DATA_BLOCK "FLT"   // DB142
{ S7_Optimized_Access := 'FALSE' }
VERSION : 0.0
// --------------------------------------------------------------------------------
//     program     :    FLT
//     description :    FLT signals       
//     name        :    G. Eibelshaeuser
//     date        :    26.10.2007
// 
//     revision    :
//     name        :
//     date        :    
//                     (c)PVA TePla AG       
//     --------------------------------------------------------------------------------
   VAR
      PD_TIME_10MBAR : Bool;   // F001 pump down time to 10 mbar exceeded
      PD_TIME_1MBAR : Bool;   // F002 pump down time to 1 mbar exceeded
      PD_TIME_01MBAR : Bool;   // F003 pump down time to 0,1 mabar exceeded
      PD_TIME_005MBAR : Bool;   // F004 pump down time to 0,05 mbar exceeded
      PD_TIME_FINAL : Bool;   // F005 pump down time to final pressure exceeded
      PD_LEAKTEST : Bool;   // F006 leaktest failed
      PD_GATE_VALVE_CLOSED : Bool;   // F007 gate valve is closed
      ME_CR_REF_POS_NOT_FND : Bool;   // F008 crucible reference position not found
      ME_LEAK_TST_FDR : Bool;   // F009 leaktest feeder failed
      ME_PRS_DROP_FDR : Bool;   // F010 pressure drop feeder too high
      ME_SPARE_F011 : Bool;   // F011
      DI_IMAGE_TO_DARK : Bool;   // F012 image too dark for dipping
      DI_TIME_CAM_EXCEEDED : Bool;   // F013 time till seed detection exceeded
      DI_TIME_MELT_EXCEEDED : Bool;   // F014 time till melt contact exceeded
      DI_SEED_NOT_CAM_STOPPED : Bool;   // F015 seed not cam. stopped before dipping
      DI_MCC_ERROR_1 : Bool;   // F016 melt contact control function error
      DI_MCC_ERROR_2 : Bool;   // F017 melt contact control input error
      DI_ISOLATION_FAULT : Bool;   // F018 crystal drive unit not isolated from ground
      DI_SPARE_F019 : Bool;   // F019
      DI_SPARE_F020 : Bool;   // F020
      NE_MAX_LEN : Bool;   // F021 max. neck length reached without constant diameter
      NE_SPARE_F022 : Bool;   // F022
      SH_MLT_LVL_SFT : Bool;   // F023 invalid melt level shift parameter in phase shoulder
      SH_SPARE_F024 : Bool;   // F024
      BY_SPARE_F025 : Bool;   // F025
      BY_SPARE_F026 : Bool;   // F026
      EC_XT_OUT_OF_MELT : Bool;   // F027 crystal out of melt
      EC_SPARE_F028 : Bool;   // F028
      EC_SPARE_F029 : Bool;   // F029
      RE_SPARE_F030 : Bool;   // F030
      RE_SPARE_F031 : Bool;   // F031
      SD_SMALL_DIS_XT_CR : Bool;   // F032 distance between crystal and crucible too small
      FDR_NOT_IN_HOME_POS : Bool;   // F033 feeder is not in home position
      CR_ROT_OSCI : Bool;   // F034 frequency of cruc. rot. oscillation too high out of range faults
      XT_ROT_OUT_OF_RNG : Bool;   // F035 crystal rotation out of range
      XT_LFT_OUT_OF_RNG : Bool;   // F036 crystal lift out of range
      CR_ROT_OUT_OF_RNG : Bool;   // F037 crucible rotation out of range
      CR_LFT_OUT_OF_RNG : Bool;   // F038 crucible lift out of range
      GAS_FLW_1_OUT_OF_RNG : Bool;   // F039 gas flow 1 out of range
      GAS_FLW_2_OUT_OF_RNG : Bool;   // F040 gas flow 2 out of range
      PRS_OUT_OF_RNG : Bool;   // F041 pressure out of range
      HTR_1_PWR_OUT_OF_RNG : Bool;   // F042 main heater power out of range
      HTR_2_PWR_OUT_OF_RNG : Bool;   // F043 bottom heater power out of range
      NECK_DIA_BELOW_LIMIT : Bool;   // F044 neck diameter below limit
      XT_GROWTH_OUT_OF_RNG : Bool;   // F045 crystal growth out of range
      XT_DIA_OUT_OF_RNG : Bool;   // F046 crystal diameter out of range
      AVG_PULL_SPD_OUT_OF_RNG : Bool;   // F047 average pull speed out of range
      MELT_LEVEL_OUT_OF_RNG : Bool;   // F048 melt level out of range
      HTR_1_RES_OUT_OF_RNG : Bool;   // F049 resistance change main heater out of range
      HTR_2_RES_OUT_OF_RNG : Bool;   // F050 resistance change bottom heater out of range
      MAG_1_CUR_OUT_OF_RNG : Bool;   // F051 magnet current coil 1 out of range
      MAG_2_CUR_OUT_OF_RNG : Bool;   // F052 magnet current coil 2 out of range
      CAM_THR_RATIO : Bool;   // F053 threshold ratio out of range from recipe temperature switches
      WTR_TMP_CUR_FEED : Bool;   // F054 water temp. current feed through heater 1
      HTR_2_TAS_CUR_FEED : Bool;   // F055 water temp. current feed through heater 2
      WTR_TMP_CR_SFT : Bool;   // F056 water temp. crucible shaft
      WTR_TMP_PWR_CAB : Bool;   // F057 water temp. high current cables
      WTR_TMP_GCH : Bool;   // F058 water temp. gate chamber
      CHAMBERS_TAS : Bool;   // F059 water temp. chambers
      VIP_TAS : Bool;   // F060 water temp. view ports
      XT_TAS : Bool;   // F061 water temp. xtal shaft
      EXH_TAS : Bool;   // F062 water temp. exhaust
      SPARE_F063 : Bool;   // F063 water flow switches -------------------
      SPARE_F064 : Bool;   // F064 spare
      WTR_FLW_HTR_1 : Bool;   // F065 water flow heater power supply
      WTR_FLW_GCH : Bool;   // F066 water flow gate chamber
      WTR_FLW_CR_SFT : Bool;   // F067 water flow crucible shaft
      XT_WFS : Bool;   // F068 water flow xtal shaft heater alarm -------------------
      HTR_SCR_WRN : Bool;   // F069 heater rectifier temp warning
      HTR_SCR_ALM : Bool;   // F070 heater rectifier temp alarm
      HTR_TRF_WRN : Bool;   // F071 heater transformer temp warning
      HTR_TRF_ALM : Bool;   // F072 heater transformer temp alarm
      THY_CTRL_1_OV_LD : Bool;   // F073 thyristor controller heater 1 overload
      THY_CTRL_1_HI_TMP : Bool;   // F074 thyristor controller heater 1 high temperature
      THY_CTRL_1_ER : Bool;   // F075 thyristor controller heater 1 fault
      HTR_2_OVERCURRENT : Bool;   // F076 heater 2 overcurrent
      HTR_2_CUR_LIMIT : Bool;   // F077 heater 2 current limit active
      HTR_2_ITL : Bool;   // F078 heater 2 interlock active UPS alarm ---------
      UPS_24V_ALM : Bool;   // F079 24 V UPS error
      UPS_24V_SPL_MIS : Bool;   // F080 24 V supply for UPS failed
      THY_CTRL_1_OV_VLT : Bool;   // F081 thryristor controller heater 1 over voltage
      CB_FLT_COMP_400V : Bool;   // F082 circuit breaker fault AC 400V compensation
      TMP_MAIN_CBT : Bool;   // F083 temperature fault main cabinet +K1 breakers and fuses ------------------
      CB_FLT_DC24V : Bool;   // F084 circuit breaker fault DC 24 V
      CB_FLT_AC230V : Bool;   // F085 circuit breaker fault AC 230 V
      CB_FLT_DRV : Bool;   // F086 circuit breaker fault drive units
      CB_FLT_AC400V : Bool;   // F087 circuit breaker fault AC 400V
      MAIN_SWITCH_OFF : Bool;   // F088 main switch of plant is off
      HTR_1_OVERCURRENT : Bool;   // F089 heater 1 overcurrent
      HTR_1_CUR_LIMIT : Bool;   // F090 heater 1 current limit active
      HTR_1_ITL : Bool;   // F091 heater 1 interlock active
      HTR_WFS : Bool;   // F092 water flow heater
      CGT_WFS : Bool;   // F093 water flow gate chamber
      CR_WFS : Bool;   // F094 water flow crucible shaft safety limit switches ---------------------
      XT_TOP_POS : Bool;   // F095 safty limit switch seed chuck in highest pos.
      XT_SLS : Bool;   // F096 safty limit switch crystal lift
      CR_SLS : Bool;   // F097 safty limit switch crucible lift
      CHAMBER_SLS : Bool;   // F098 safty limit switch chamber lift
      MAG_SLS : Bool;   // F099 safty limit switch magnet lift
      MAIN_LINE_460V_OFF : Bool;   // F100 460V main power supply is off image processing unit ---------------------
      INIT_FLT_IM_PROC_UNIT : Bool;   // F101 initialisation fault image processing unit
      INV_DATA_IM_PROC_UNIT : Bool;   // F102 invalid data from image processing unit
      CAM_INTERFACE_INIT : Bool;   // F103 camera serial interface init failed
      CAM_THR_ADJ_STOPPED : Bool;   // F104 automatic threshold adjustment interrupted
      CAM_THR_ADJ_ABORTED : Bool;   // F105 automatic threshold adjustment aborted common ------
      MAIN_LINE_OFF : Bool;   // F106 main power supply is off
      COM_AIR_PRS_LOW : Bool;   // F107 compressed air pressure is below limit
      PLC_INIT_FLT_NO_RECIPE : Bool;   // F108 no recipe in PLC
      EMO : Bool;   // F109 emergency off
      DRV_CAL_MIS : Bool;   // F110 drive calibration is missing
      LSR_RCV : Bool;   // F111 laser receiver detects no beam drive controller faults
      DRV_XT_LFT_PAR_FLT : Bool;   // F112 parameter fault drive controller crystal lift
      DRV_XT_LFT_RUN_FLT : Bool;   // F113 operating fault drive controller crystal lift
      DRV_XT_ROT_PAR_FLT : Bool;   // F114 parameter fault drive controller crystal rotation
      DRV_XT_ROT_RUN_FLT : Bool;   // F115 operating fault drive controller crystal rotation
      DRV_CR_LFT_PAR_FLT : Bool;   // F116 parameter fault drive controller crucible lift
      DRV_CR_LFT_RUN_FLT : Bool;   // F117 operating fault drive controller crucible lift
      DRV_CR_ROT_PAR_FLT : Bool;   // F118 parameter fault drive controller crucible rotation
      DRV_CR_ROT_RUN_FLT : Bool;   // F119 operating fault drive controller crucible rotation
      DRV_CHB_LFT_PAR_FLT : Bool;   // F120 parameter fault drive controller chamber lift
      DRV_CHB_LFT_RUN_FLT : Bool;   // F121 operating fault drive controller chamber lift
      DRV_CHB_SW_PAR_FLT : Bool;   // F122 parameter fault drive controller chamber swivel
      DRV_CHB_SW_RUN_FLT : Bool;   // F123 operating fault drive controller chamber swivel
      SPARE_F124 : Bool;   // F124
      WTR_TMP_CFT_2 : Bool;   // F125 water temperature current feed throughs 2
      WTR_TMP_GATE : Bool;   // F126 water temperature gate and gate valve
      WTR_TMP_SPC : Bool;   // F127 water temperature spacer and view ports
      WTR_TMP_VSL : Bool;   // F128 water temperature vessel parts Vacuum faults --------------------
      P1 : Bool;   // F129 vacuum pump 1 not ready
      P2 : Bool;   // F130 vacuum pump 2 not ready
      P3 : Bool;   // F131 vacuum pump 3 not ready
      P1_TMP_HIGH : Bool;   // F132 temperature fault of pump 1
      P2_TMP_HIGH : Bool;   // F133 temperature fault of pump 2
      P3_TMP_HIGH : Bool;   // F134 temperature fault of pump 3
      V7 : Bool;   // F135 undefined position gate valve
      V2_1 : Bool;   // F136 vacuum valve V2.1 not open
      V2_2 : Bool;   // F137 vacuum valve V2.2 not open
      V3 : Bool;   // F138 vacuum valve V3 not open
      WTR_TMP_FCH : Bool;   // F139 water temperature furnace chamber
      WTR_TMP_TCH : Bool;   // F140 water temperature top chamber
      P1_SP_WRN : Bool;   // F141 vacuum pump 1 warning active
      FDR_HOP_NOT_CON : Bool;   // F142 hopper not connected to feeder
      P3_SP_WRN : Bool;   // F143 vacuum pump 3 warning active
      WTR_FLW_FCH : Bool;   // F144 water flow furnace chamber
      WTR_FLW_TCH : Bool;   // F145 water flow top chamber
      WTR_FLW_CFT_2 : Bool;   // F146 water flow current feed throughs 2
      WTR_FLW_GATE : Bool;   // F147 water flow gate and gate valve
      WTR_FLW_SPC : Bool;   // F148 water flow spacer and view ports
      WTR_FLW_VSL : Bool;   // F149 water flow bottom chamber Position encoder faults -----------------------
      ENC_XT_LFT : Bool;   // F150 position error crystal lift
      ENC_CR_LFT : Bool;   // F151 position error crucible lift
      ENC_CGT_LFT : Bool;   // F152 position error handling lift
      SPARE_F153 : Bool;   // F153 image processing with DVT Cam -----------------------------
      CAM_ROI_OUTSIDE : Bool;   // F154 camera measurement area is outside the image frame
      DVT_PRD_NO_PLC : Bool;   // F155 Produktnummer in der SPS ung黮tig
      DVT_PRD_NO_IMG_SEN : Bool;   // F156 Produktnummer in Kamera ist ung黮tig
      CAM_COM_SEND : Bool;   // F157 Sendefehler SPS - Kamera
      CAM_DATA_RECV : Bool;   // F158 Empfangsfehler SPS - Kamera
      DVT_NO_PRD : Bool;   // F159 kein "P" im Telegramm von Kamera
      DVT_DATA_MSG : Bool;   // F160 Daten von Kamera sind ung黮tig
      DVT_PRD_NO_DIF : Bool;   // F161 Produktnummer von Kamera ist falsch
      CAM_NDR_TOUT : Bool;   // F162 keine Daten von Kamera empfangen
      DVT_IMG_SEN : Bool;   // F163 Bildverarbeitung von Kamera gescheitert
      CAM_NO_CTR_FND : Bool;   // F164 Kamera findet keinen messbaren Kontrast
      CAM_MSR_INSTAB : Bool;   // F165 Meniskusmessung instabil, Fehlmessungen -----------------------
      V7_CLOSED : Bool;   // F166 gate valve closed (crystal down disabled)
      CLF_CLP_POS : Bool;   // F167 undefined position furnace clamp
      CGT_COUPLE : Bool;   // F168 undefined position coupling gate/furnace
      CLF_SWL_POS : Bool;   // F169 undefined position lower furnace
      HND_VACUUM : Bool;   // F170 furnace is not vented !
      CLF_CLAMP : Bool;   // F171 upper furnace is not connected with gate !
      XT_FORK : Bool;   // F172 safety fork installed (crystal down disabled)
      SEED_TMP : Bool;   // F173 seed chuck is too hot; crystal lift stopped
      FDR_TUBE_TME_OUT : Bool;   // F174 feeding tube did not reach end position
      GCH_NOT_CL : Bool;   // F175 gate chamber not closed
      CR_ROT_CAL : Bool;   // F176 calibration fault crucible rotation drive
      CR_LFT_CAL : Bool;   // F177 calibration fault crucible lift drive
      XT_ROT_CAL : Bool;   // F178 calibration fault crystal rotation drive
      XT_LFT_CAL : Bool;   // F179 calibration fault crystal lift drive
      WTR_FLW_PLT : Bool;   // F180 water flow chamber parts and view ports
      PWR_SPL_WFS : Bool;   // F181 water flow heater power supply
      WTR_FLW_CUR_FEED : Bool;   // F182 water flow current feed through heater 1
      WTR_FLW_PWR_CAB : Bool;   // F183 water flow high current cables
      WTR_FLW_GCH_V : Bool;   // F184 water flow gate chamber valve
      WTR_FLW_CONE : Bool;   // F185 water flow cone alarm /nur SC22 AUO)
      WTR_TMP_PLT : Bool;   // F186 water temp. chamber parts and view ports
      WTR_TMP_GCH_V : Bool;   // F187 water temp. gate chamber valve
      WTR_TMP_HTR_1 : Bool;   // F188 water temp. heater power supply
      PWR_SPL_INT_TAS : Bool;   // F189 water temp. transformer intern
      WTR_TMP_HIGH_LIM : Bool;   // F190 water temp. high limit reached
      HTR_PWR_CAB_TAS : Bool;   // F191 water temp. high power cables
      HTR_1_TAS_CUR_FEED : Bool;   // F192 water temp. current feed through heater 1
      CGT_TAS : Bool;   // F193 water temp. gate chamber
      CR_TAS : Bool;   // F194 water temp. crucible shaft MAGNET FAULTS -------------
      MAG_1_RES_OUT_OF_RNG : Bool;   // F195 resistance change upper magnet out of range
      MAG_2_RES_OUT_OF_RNG : Bool;   // F196 resistance change lower magnet out of range
      MAG_WFS : Bool;   // F197 water flow magnet power supply intern
      MAG_1_ITL : Bool;   // F198 magnet 1 rectifier interlock active
      MAG_2_ITL : Bool;   // F199 magnet 2 rectifier interlock active
      MAG_TMP_ALM : Bool;   // F200 magnet transformer temperature alarm
      MAG_1_EXT_ITL : Bool;   // F201 external interlock magnet 1
      MAG_2_EXT_ITL : Bool;   // F202 external interlock magnet 2
      MAG_DOOR_ITL : Bool;   // F203 door interlock magnet power supply
      MAG_1_OVERCURRENT : Bool;   // F204 magnet 1 overcurrent
      MAG_2_OVERCURRENT : Bool;   // F205 magnet 2 overcurrent
      PAR_FLT_MAG_1_CUR : Bool;   // F206 magnet 1 current setpoint out of range
      PAR_FLT_MAG_2_CUR : Bool;   // F207 magnet 2 current setpoint out of range
      MAG_LFT_SDL_ERR : Bool;   // F208 Magnet lift error - upward lift disabled
      MAG_TAS : Bool;   // -----------------
      DP_ADR_08_NOT_PRESENT : Bool;   // F210 dp-slave not present (+N2)
      DP_ADR_09_NOT_PRESENT : Bool;   // F211 dp-slave not present (+R1.B1)
      DP_ADR_10_NOT_PRESENT : Bool;   // F212 dp-slave not present (+N1)
      DP_ADR_11_NOT_PRESENT : Bool;   // F213 dp-slave not present (+N4)
      DP_ADR_16_NOT_PRESENT : Bool;   // F214 dp-slave encoder crystal lift not present
      DP_ADR_17_NOT_PRESENT : Bool;   // F215 dp-slave encoder crucible lift not present
      DP_ADR_18_NOT_PRESENT : Bool;   // F216 dp-slave encoder handling lift not present
      DP_ADR_32_NOT_PRESENT : Bool;   // F217 dp-slave controller crystal rot. not present
      DP_ADR_33_NOT_PRESENT : Bool;   // F218 dp-slave controller crystal lift not present
      DP_ADR_34_NOT_PRESENT : Bool;   // F219 dp-slave controller crucible rot. not present
      DP_ADR_35_NOT_PRESENT : Bool;   // F220 dp-slave controller crucible lift not present
      DP_ADR_36_NOT_PRESENT : Bool;   // F221 dp-slave controller gate swinging not present
      DP_ADR_37_NOT_PRESENT : Bool;   // F222 dp-slave controller gate lifting not present
      DP_ADR_40_NOT_PRESENT : Bool;   // F223 dp-slave main heater not present
      DP_ADR_41_NOT_PRESENT : Bool;   // F224 dp-slave botton heater not present
      DP_ADR_45_NOT_PRESENT : Bool;   // F225 dp-slave magnet coil 1 not present
      DP_ADR_46_NOT_PRESENT : Bool;   // F225 dp-slave magnet coil 2 not present
      DP_ADR_64_NOT_PRESENT : Bool;   // F227 dp-slave not present (+N5)
      DP_ADR_13_NOT_PRESENT : Bool;   // F228 dp-slave not present (+N3)
      DP_ADR_48_NOT_PRESENT : Bool;   // F229 dp-slave MFC 1 not present
      DP_ADR_42_NOT_PRESENT : Bool;   // F230 dp-slave SCR controller heater 1 not present
      DP_ADR_43_NOT_PRESENT : Bool;   // F231 dp-slave SCR controller heater 2 not present
      DP_ADR_38_NOT_PRESENT : Bool;   // F232 dp_slave pump unit not present
      DP_ADR_08_ERROR : Bool;   // F233 dp-slave fault (+N1)
      DP_ADR_09_ERROR : Bool;   // F234 dp-slave fault (+R1.B1)
      DP_ADR_10_ERROR : Bool;   // F235 dp-slave fault (+N2)
      DP_ADR_11_ERROR : Bool;   // F236 dp-slave fault (+N4)
      DP_ADR_16_ERROR : Bool;   // F237 dp-slave encoder crystal lift fault
      DP_ADR_17_ERROR : Bool;   // F238 dp-slave encoder crucible lift fault
      DP_ADR_18_ERROR : Bool;   // F239 dp-slave encoder handling lift fault
      DP_ADR_32_ERROR : Bool;   // F240 dp-slave controller crystal rot. fault
      DP_ADR_33_ERROR : Bool;   // F241 dp-slave controller crystal lift fault
      DP_ADR_34_ERROR : Bool;   // F242 dp-slave controller crucible rot. fault
      DP_ADR_35_ERROR : Bool;   // F243 dp-slave controller crucible lift fault
      DP_ADR_36_ERROR : Bool;   // F244 dp-slave controller gate swinging fault
      DP_ADR_37_ERROR : Bool;   // F245 dp-slave controller gate lifting fault
      DP_ADR_40_ERROR : Bool;   // F246 dp-slave main heater fault
      DP_ADR_41_ERROR : Bool;   // F247 dp-slave bottom heater fault
      DP_ADR_45_ERROR : Bool;   // F248 dp-slave magnet coil 1 fault
      DP_ADR_46_ERROR : Bool;   // F249 dp-slave magnet coil 2 fault
      DP_ADR_64_ERROR : Bool;   // F250 dp-slave fault (+N5)
      DP_ADR_13_ERROR : Bool;   // F251 dp-slave fault (+N3)
      DP_ADR_48_ERROR : Bool;   // F252 dp-slave MFC 1 fault
      DP_ADR_42_ERROR : Bool;   // F253 dp-slave SCR controller heater 1 fault
      DP_ADR_43_ERROR : Bool;   // F254 dp-slave SCR controller heater 2 fault
      DP_ADR_38_ERROR : Bool;   // F255 dp-slave pump unit fault
      SPARE_F256 : Bool;   // F256 device faults -------------
      MSR_WTR_TMP_PWR_CAB : Bool;   // F257 measurement water temp. high current cables
      MSR_WTR_FLW_PWR_CAB : Bool;   // F258 measurement water flow high current cables
      MSR_WTR_TMP_CUR_FEED : Bool;   // F259 measurement water temp. cur. feed through 1
      MSR_WTR_FLW_CUR_FEED : Bool;   // F260 measurement water flow cur. feed through 1
      MSR_WTR_TMP_CR_SFT : Bool;   // F261 measurement water temp. crucible shaft
      MSR_WTR_FLW_CR_SFT : Bool;   // F262 measurement water flow crucible shaft
      MSR_WTR_TMP_HTR_1 : Bool;   // F263 measurement water temp. heater 1 power supply
      MSR_WTR_FLW_HTR_1 : Bool;   // F264 measurement water flow heater 1 power supply
      MSR_WTR_TMP_CFT_2 : Bool;   // F265 measurement water temp. cur.feed through 2
      MSR_WTR_FLW_CFT_2 : Bool;   // F266 measurement water flow cur. feed through 2
      MSR_WTR_TMP_GATE : Bool;   // F267 measurement water temp. gate and gate valve
      MSR_WTR_FLW_GATE : Bool;   // F268 measurement water flow gate and gate valve
      MSR_WTR_TMP_SPC : Bool;   // F269 measurement water temp. spacer and view ports
      MSR_WTR_FLW_SPC : Bool;   // F270 measurement water flow spacer and view ports
      MSR_WTR_TMP_VSL : Bool;   // F271 measurement water temp. bottom chamber
      MSR_WTR_FLW_VSL : Bool;   // F272 measurement water flow bottom chamber
      MSR_WTR_TMP_FCH : Bool;   // F273 measurement water temp. furnace chamber
      MSR_WTR_FLW_FCH : Bool;   // F274 measurement water flow furnace chamber
      MSR_WTR_TMP_TCH : Bool;   // F275 measurement water temp. top chamber
      MSR_WTR_FLW_TCH : Bool;   // F276 measurement water flow top chamber
      MSR_ACT_MLT_TMP : Bool;   // F277 measurement melt temperature
      MSR_ACT_HTR_1_TMP : Bool;   // F278 measurement heater 1 temperature
      MLT_TMP_SIG : Bool;   // F279 melt temperature signal not valid
      HTR_1_TMP_SIG : Bool;   // F280 heater 1 temperature signal not valid
      MSR_P1_VIB : Bool;   // F281 measurement screw pump P1 vibration
      V25 : Bool;   // F282 fault valve 25
      XT_DRP_OUT_PRT_OP : Bool;   // F283 crystal drop out protection not opened
      XT_DRP_OUT_PRT_CL : Bool;   // F284 crystal drop out protection not closed
      HTR_1_SCR_ALM : Bool;   // F285 heater 1 rectifier temp alarm
      HTR_1_TRF_WRN : Bool;   // F286 heater 1 transformer temp warning
      HTR_1_TRF_ALM : Bool;   // F287 heater 1 transformer temp alarm
      HTR_2_SCR_ALM : Bool;   // F288 heater 2 rectifier temp alarm
      HTR_2_TRF_WRN : Bool;   // F289 heater 2 transformer temp warning
      HTR_2_TRF_ALM : Bool;   // F290 heater 2 transformer temp alarm
      THY_CTRL_2_OV_LD : Bool;   // F291 thyristor controller heater 2 overload
      THY_CTRL_2_HI_TMP : Bool;   // F292 thyristor controller heater 2 high temperature
      THY_CTRL_2_ER : Bool;   // F293 thyristor controller heater 2 fault
      THY_CTRL_2_OV_VLT : Bool;   // F294 thryristor controller heater 2 over voltage
      MSR_WTR_TMP_PLT : Bool;   // F295 measurement water temp. vessel and view ports
      MSR_WTR_FLW_PLT : Bool;   // F296 measurement water flow vessel and view ports
      MSR_WTR_TMP_GCH : Bool;   // F297 measurement water temp. gate chamber
      MSR_WTR_FLW_GCH : Bool;   // F298 measurement water flow gate chamber
      MSR_WTR_TMP_GCH_V : Bool;   // F299 measurement water temp. gate chamber valve
      MSR_WTR_FLW_GCH_V : Bool;   // F300 measurement water flow gate chamber valve
      V15 : Bool;   // F301 fault valve 15
      V14 : Bool;   // F302 fault valve 14
      V12 : Bool;   // F303 fault valve 12
      V18 : Bool;   // F304 fault valve 18
      V17 : Bool;   // F305 fault valve 17
      V13 : Bool;   // F306 fault valve 13
      P1_GEAR_OIL_TMP_WRN : Bool;   // F307 warning gear oil temperature of screw pump P1
      P1_GEAR_OIL_TMP_ALM : Bool;   // F308 alarm gear oil temperature of screw pump P1
      P1_COOLANT_TMP_WRN : Bool;   // F309 warning coolant temperature of screw pump P1
      P1_COOLANT_TMP_ALM : Bool;   // F310 alarm coolant temperature of screw pump P1
      DP_ADR_50_NOT_PRESENT : Bool;   // F311 dp_slave Simocode P1 not present
      DP_ADR_51_NOT_PRESENT : Bool;   // F312 dp_slave Simocode P2 not present
      DP_ADR_50_ERROR : Bool;   // F313 dp-slave Simocode P1 fault
      DP_ADR_51_ERROR : Bool;   // F314 dp-slave Simocode P2 fault
      FSH_MAIN_SI_FIL : Bool;   // F315 flushing of main Si filter not done
      FSH_AUX_SI_FIL : Bool;   // F316 flushing of aux Si filter not done
      WTR_TMP_VPTS : Bool;   // F317 water temperature view ports
      WTR_FLW_VPTS : Bool;   // F318 water flow view ports
      P1_VIB_ALM : Bool;   // F319 vibration of Pump 1 above alarm level
      MSR_P1_PT100_GEAR_OIL : Bool;   // F320 measurement error of PT100 sensor P1 gear oil temp.
      MSR_P1_PT100_COOLANT : Bool;   // F321 measurement error of PT 100 sensor P1 coolant temp.
      INIT_KL_3202 : Bool;   // F322 Initialisation of PT 100 terminal failed (KL3202)
      MSR_WTR_TMP_VPTS : Bool;   // F323 measurement water temperature view ports
      MSR_WTR_FLW_VPTS : Bool;   // F324 measurement water flow view ports
      PHA_CUR_P1 : Bool;   // F325 phase current of Pump 1 above limit
      PHA_CUR_P2 : Bool;   // F326 phase current of Pump 2 above limit
      CR_LFT_NO_ROT : Bool;   // F327 crucible lift without shaft rotation
      INGOT_ID_TIME_OUT : Bool;   // F328 timeout ingot ID
      CARRIER_ID_REFUSED : Bool;   // F329 carrier ID refused from MES
      XT_ORB_ABV_LIM : Bool;   // F330 crystal orbiting is above limit
      PU_WRN : Bool;   // F331 pump unit warning
      PU_ERR : Bool;   // F332 pump unit error
      DST_MLT_FNL_SML : Bool;   // F333 distance melt level to funnel too small
      DST_MLT_FNL_LRG : Bool;   // F334 distance metl level to funnel too large
      MLT_LVL_MSR_NOT_VALID : Bool;   // F335 melt level measurements not valid - control loop switched off
      XT_LFT_SW_LIMIT : Bool;   // F336 software limitation of crystal lift is reached
      CR_LFT_SW_LIMIT : Bool;   // F337 software limitation of crucible lift is reached
      HTR_1_PWR_SPL : Bool;   // F338 heater 1 power supply fault
      HTR_1_PWR_SPL_WRN : Bool;   // F339 heater 1 power supply warning
      HTR_1_PWR_SPL_IN_LOC : Bool;   // F340 heater 1 power supply in local operation mode
      MSR_CGT_BAR_ACT_PRS_1000 : Bool;   // F341 measurement vacuum gauge gate chamber
      OV_VLT_PRT : Bool;   // F342 over-voltage protection fault in main line
      HTR_1_BUS_BAR_TMP : Bool;   // F343 high bus bar temperature of heater 1 power supply
      HTR_2_BUS_BAR_TMP : Bool;   // F344 high bus bar temperature of heater 2 power supply
      MSR_WTR_FLW_PU : Bool;   // F345 measurement water flow pump unit
      MSR_WTR_TMP_PU : Bool;   // F346 measurement water temperature pump unit
      CAM_DI_XT_DN_ARB : Bool;   // F347 camera controlled seed down off - crystal speed reduced
      CAM_HTR_1_IN_SMI : Bool;   // F348 growth control off - heater 1 switched to semi automatic
      CAM_CRUC_ROT_IN_SMI : Bool;   // F349 growth control off - crucible rotation switched to semi automatic
      CAM_DIA_CTRL_OFF : Bool;   // F350 diameter control off - crystal lift switched to semi automatic
      WTR_TMP_PU : Bool;   // F351 water temperature pump unit
      SI_FIL_REG_ENB : Bool;   // F352 filter regeneration is not enabled and aborted
      INIT_KL2552 : Bool;   // F353 initialisation of gate chamber swivel controller failed
      MSR_TRV_ACT_POS : Bool;   // F354 measurement actual control valve position
      COOL_UNIT_CAB : Bool;   // F355 fault cooling unit of cabinet
      V3_0 : Bool;   // F356 vacuum valve V3.0 in undefined position
      V3_1 : Bool;   // F357 vacuum valve V3.1 in undefined position
      MOB_FDR_CB_AC_230V : Bool;   // F358 circuit breaker fault AC230V of mobile feeder
      MOB_FDR_CB_DC_24V : Bool;   // F359 circuit breaker fault AC24V of mobile feeder
      XT_LFT_POS_REF : Bool;   // F360 position reference of crystal lift encoder is missing
      CR_LFT_POS_REF : Bool;   // F361 position reference of crucible lift encoder is missing
      HND_COL_GCH_TCH : Bool;   // F362 collision warning gate chamber - top chamber
      HND_COL_TCH_FCH : Bool;   // F363 collision warning top chamber - furnace chamber
      MOB_FDR_INIT_KL_3312 : Bool;   // F364 initialisation of feeder temperature measurement failed
      MOB_FDR_TC_TUBE : Bool;   // F365 thermocouple feeder tube failed
      MOB_FDR_INIT_KL2552 : Bool;   // F366 initialisation of mobile feeder drive controller failed
      ECS_UG_NOT_LD : Bool;   // F367 DC voltage source of drive controllers not available
      MOB_FDR_MOV_IN_SEQ_ABR : Bool;   // F368 tube move in sequence of mobile feeder aborted
      MOB_FDR_MOV_OUT_SEQ_ABR : Bool;   // ----------------------------
      DAG_STARTUP : Bool;   // F370 DAG Startup calibration
      DAG_AC : Bool;   // F371 DAG AC extern
      DAG_SHRT_CRCT : Bool;   // F372 DAG short circuit
      DAG_HIGH_TMP : Bool;   // F373 DAG high temperatur
      DAG_DC_INT : Bool;   // F374 DAG DC intern
      DAG_OVERLOAD : Bool;   // F375 DAG overload over 1min Magnet EKZ 3500 ---------------
      MAG_PWR_SPL : Bool;   // F376 Power supply of magnet failed
      MAG_QUENCH : Bool;   // F377 Quench failure of magnet
      MAG_EMG_OFF : Bool;   // F378 Emergency shut down of magnet
      MAG_MAIN_LINE : Bool;   // F379 Main line failure of magnet
      MAG_TMP : Bool;   // F380 Temperature of magnet is too high
      MAG_CUR_FEED : Bool;   // F381 Voltage failure of magnet
      MAG_VAC : Bool;   // F382 Vacuum failure of magnet
      MAG_HE_COMPR : Bool;   // F383 He-Compressor of magnet failed
      WRN_MAG : Bool;   // F384 Warning magnet
      WTR_TMP_CONE : Bool;   // F385 Cooling water temperature cone high (nur SC22 - AUO)
      WRN_UPR_CR_POS_LIM : Bool;   // F386 Warning distance melt level to funnel reached
      ALM_UPR_CR_POS_LIM : Bool;   // F387 Alarm distance melt level to funnel reached - crucible stopped
      CB_CAP_BOX_HTR1 : Bool;   // F388 circuit breaker fault AC 400V capacitor htr1
      CB_CAP_BOX_HTR2 : Bool;   // F389 circuit breaker fault AC 400V capacitor htr2 Aktivk黨lung -------------
      DIST_MELT_FUN : Bool;   // F390 ACC: distance melt level to funnel is too low
      MSR_ACC_WTR_TMP : Bool;   // F391 ACC: measurement water outlet temperature in cooling coil
      MSR_ACC_WTR_PRS_IN : Bool;   // F392 ACC: measurement water pressure in cooling coil
      MSR_ACC_WTR_FLW_OUT : Bool;   // F393 ACC: measurement water outlet flow in cooling coil
      MSR_ACC_WTR_FLW_IN : Bool;   // F394 ACC: measurement water inlet flow in cooling coil
      ACC_WRN_WTR_TMP : Bool;   // F395 ACC: water outlet temp. in cooling coil above warning limit
      ACC_WRN_WTR_PRS_IN : Bool;   // F396 ACC: water pressure in cooling coil below limit
      ACC_WRN_WTR_FLW_OUT : Bool;   // F397 ACC: water outlet flow in cooling coil below warning limit
      ACC_WRN_WTR_FLW_IN : Bool;   // F398 ACC: water inlet flow in cooling coil below warning limit
      ACC_CB_FLT_DC24V : Bool;   // F399 ACC: circuit breaker fault DC 24V
      ACC_WRN_FCH_OV_PRS_1 : Bool;   // F400 ACC: furnace overpressure detected at switch 1
      ACC_WRN_FCH_OV_PRS_2 : Bool;   // F401 ACC: furnace overpressure detected at switch 2
      ACC_UPS_BAT_MODE : Bool;   // F402 ACC: 24V UPS is in battery mode
      ACC_UPS_24V_ALM : Bool;   // F403 ACC: 24V UPS fault
      ACC_SC_WTR : Bool;   // F404 ACC: safety circuit cooling water tripped
      ACC_SC_HTR : Bool;   // F405 ACC: safety circuit heater tripped
      ACC_WRN_WTR_SPL_PRS : Bool;   // F406 ACC: water supply pressure below limit
      MSR_ACC_WTR_SPL_PRS : Bool;   // F407 ACC: measurement water supply pressure
      ACC_EXH_FLP_CLD : Bool;   // F408 ACC: over pressure flap not closed
      ACC_WTR_FLW_IN : Bool;   // F409 ACC: water inlet flow in cooling coil too low
      ACC_WTR_FLW_OUT : Bool;   // F410 ACC: water outlet flow in cooling coil too low
      ACC_WTR_TMP_OUT : Bool;   // F411 ACC: water outlet temperature in cooling coil too high
      ACT_WTR_TMP_RING : Bool;   // F412 ACC: water temperature in spacer flange too high
      ACT_WTR_FLW_RING : Bool;   // F413 ACC: water flow in spacer flange too low
      ACC_OVP_TEST : Bool;   // F414 ACC: overpressure test failed
      ACC_TC : Bool;   // F415 ACC: water temp. in cooling coil above warn. limit (TC)
      MAKE_OVP_TEST : Bool;   // F416 ACC: overpressure test not done
      ACC_WTR_DIFF : Bool;   // F417 ACC: water flow deviation in cooling coil between inlet and outlet
      ACT_WTR_TMP_WARN : Bool;   // F418 ACC: water temperature in spacer flange above warning limit
      ACC_EX_ALARM : Bool;   // F419 ACC: danger - unexpected pressure rise in furnace
      MOB_FDR_DP_ERROR : Bool;   // F420 dp-slave fault of mobile feeder
      MOB_FDR_DP_NOT_PRESENT : Bool;   // F421 dp-slave of mobile feeder not present
      MOB_FDR_NOT_DCK : Bool;   // F422 mobile feeder not docked to puller
      MOB_FDR_STP_PARA : Bool;   // F423 step parameters of feeder are not valid
      MOB_FDR_DCK_SEQ_ABR : Bool;   // F424 docking sequence of mobile feeder aborted
      MOB_FDR_UDCK_SEQ_ABR : Bool;   // F425 undocking sequence of mobile feeder aborted
      MOB_FDR_FNC_PRS_HI : Bool;   // F426 furnace pressure too high for leak test of feeder valve
      MOB_FDR_PRS_HI : Bool;   // F427 feeder pressure too high for leak test of feeder valve
      HTR_2_PWR_SPL : Bool;   // F428 heater 2 power supply fault
      HTR_2_PWR_SPL_WRN : Bool;   // F429 heater 2 power supply warning
      HTR_2_PWR_SPL_IN_LOC : Bool;   // F430 heater 2 power supply in local operation mode
      ACC_OVP_1_FLT : Bool;   // F431 ACC: overpressure switch 1 failed
      ACC_OVP_2_FLT : Bool;   // F432 ACC: overpressure switch 2 failed
      ME_MLT_TMP_TOO_HI : Bool;   // F433 melt temperature too high
      FEED_RTE_TOO_HI : Bool;   // F434 feed rate too high
      XT_MEN_CNTR : Bool;   // F435 crystal meniscus contracted - diameter control off
      HTR_1_HOT_RES : Bool;   // F436 hot resistance main heater out of range
      ACC_CB_FLT_AC230V : Bool;   // F437 ACC: circuit breaker fault AC 230 V
      ACC_WTR_PRS_COMP_TANK : Bool;   // F438 ACC: diaphragm of cooling water compensation tank failed
      ACC_DP_ERROR : Bool;   // F439 ACC: dp-slave fault of active cooling
      ACC_DP_NOT_PRESENT : Bool;   // F440 ACC: dp-slave of active cooling not present
      SI_FIL_NOT_VENTED : Bool;   // F441 exhaust filter is not vented
      DST_MLT_FNL_TOO_LOW : Bool;   // F442 highest crucible position reached
      DP_ADR_14_NOT_PRESENT : Bool;   // F443 dp-slave not present (+N7)
      DP_ADR_14_ERROR : Bool;   // F444 dp-slave fault (+N7)
      V1_POS_EXC_LWR_LIM : Bool;   // F445 actual V1 position falls below lower limit
      V1_POS_EXC_UPR_LIM : Bool;   // F446 actual V1 position exceeds upper limit
      V21_NOT_OPEN : Bool;   // F447 V21 is not open - release conditions are not met
      MSR_WTR_TMP_ACC_FLG : Bool;   // F448 ACC: measurement water temperature ACC flange
      MSR_WTR_FLW_ACC_FLG : Bool;   // F449 ACC: measurement water flow ACC flange
      EMO_P1 : Bool;   // F450 emergency off vacuum pump P1
      FIL_REG_NOT_DONE : Bool;   // F451 filter regeneration is not done
      GATE_V_NOT_CLD : Bool;   // F452 gate valve is not closed
      MOB_FDR_PMP_TME : Bool;   // F453 Feeder final pressure not reached pumping time to long
      MOB_FDR_VIB_SET_P_ALM : Bool;   // F454 Set point of feed rate control exceeds limitation
      DEV_ERR_WTR_TCH : Bool;   // F455 Device error, Water flow top chamber
      DEV_ERR_WTR_PWR_CAB : Bool;   // F456 Device error, Water flow high current cables
      DEV_ERR_WTR_FCH : Bool;   // F457 Device error, Water flow furnace chamber
      DEV_ERR_WTR_PU : Bool;   // F458 Device error, Water flow pump unit
      DEV_ERR_WTR_GCH_VSL : Bool;   // F459 Device error, Water flow bottom chamber
      DEV_ERR_WTR_GCH_V : Bool;   // F460 Device error, Water flow gate chamber valve
      DEV_ERR_WTR_HTR_1 : Bool;   // F461 Device error, Water flow heater power supply
      DEV_ERR_WTR_CR_SFT : Bool;   // F462 Device error, Water flow crucible shaft
      DEV_ERR_WTR_GCH : Bool;   // F463 Device error, Water flow gate chamber
      DEV_ERR_WTR_CUR_FED : Bool;   // F464 Device error, Water flow current feed through heater 1
      DEV_ERR_WTR_CFT_2 : Bool;   // F465 Device error, Water flow current feed through heater 2
      DEV_ERR_WTR_VPTS : Bool;   // F466 Device error, Water flow temperature view ports
      DEV_ERR_WTR_XT_SFT : Bool;   // F467 Device error, water flow seed shaft
      DEV_ERR_WTR_GCH_H : Bool;   // F468 Device error, water flow gate chamber valve housing
      DEV_ERR_WTR_TEC_FLG : Bool;   // F469 Device error, water flow technolity chamber
      DEV_ERR_WTR_UP_FCH : Bool;   // F470 Device error, water flow upper furnace chamber
      DEV_ERR_WTR_BCH : Bool;   // F471 Device error, water flow bottom chamber
      DEV_ERR_WTR_SOC_BCH : Bool;   // F472 Device error, water flow socket bottom chamber
      DEV_ERR_WTR_PWR_CAB2 : Bool;   // F473 Device error, water flow high current cables heater 2
      DEV_ERR_WTR_ACC : Bool;   // F474 Device error, water flow active cooling
      DEV_ERR_WTR_GCH_ADDS : Bool;   // F475 Device error, water flow gate chamber additions
      DEV_ERR_WTR_MAG_CO1 : Bool;   // F476 Device error, water flow magnet compressor unit 1
      DEV_ERR_WTR_MAG_CO2 : Bool;   // F477 Device error, water flow magnet compressor unit 2
      DEV_ERR_WTR_MAG_CO3 : Bool;   // F478 Device error, water flow magnet compressor unit 3
      DEV_ERR_WTR_MAG_CO4 : Bool;   // F479 Device error, water flow magnet compressor unit 4
      DEV_ERR_WTR_MAG_CAB : Bool;   // F480 Device error, water flow magnet power supply
      DEV_ERR_WTR_HLD_ACC : Bool;   // F481 Device error, water flow holder active cooling
      DEV_ERR_WTR_VAC_BYP : Bool;   // F482 Device error, water flow vacuum bypass tube
      SPARE_F483 : Bool;   // F483
      PN_COM_PLC : Bool;   // F484 Profinet network error PLC
      PN_COM : Bool;   // F485 Profinet IO is not Working
      PN_COM_XT_LFT_DRV : Bool;   // F486 Profinet network error, xtal-lift drive
      PN_COM_XT_ROT_DRV : Bool;   // F487 Profinet network error,,xtal-rot drive
      PN_COM_CR_LFT_DRV : Bool;   // F488 Profinet network error, crucible-lift drive
      PN_COM_CR_ROT_DRV : Bool;   // F489 Profinet network error,,crucible-rot drive
      PN_COM_HND_LFT_DRV : Bool;   // F490 Profinet network error, handling lift drive
      PN_COM_DEZ_IO_1 : Bool;   // F491 Profinet network error, Device decentral I-O
      PN_COM_HTR_1 : Bool;   // F492 Profinet network error, Heater 1
      PN_COM_HTR_2 : Bool;   // F493 Profinet network error, Heater 2
      PN_COM_MFC_1 : Bool;   // F494 Profinet network error, MFC 1
      PN_COM_MFC_2 : Bool;   // F495 Profinet network error, MFC 2
      PN_COM_HND_LFT_ENC : Bool;   // F496 Profinet network error, handling lift drive
      PN_COM_IO_MASTER_WTR_1 : Bool;   // F497 Profinet network error, IO-LINK Master 1
      PN_COM_IO_MASTER_WTR_2 : Bool;   // F498 Profinet network error, IO-Link Master 2
      PN_COM_IO_MASTER_WTR_3 : Bool;   // F499 Profinet network error, IO-Link Master 3
      PN_COM_IO_MASTER_WTR_4 : Bool;   // F500 Profinet network error, IO-Link Master 4
      PN_COM_SWITCH_1 : Bool;   // F501 Profinet network error, Switch 1
      PN_COM_SWITCH_2 : Bool;   // F502 Profinet network error, Switch 2
      PN_COM_SWITCH_3 : Bool;   // F503 Profinet network error, Switch 3
      PN_COM_TEC_FLG_LFT_DRV : Bool;   // F504 Profinet network error technology flange lift drive
      PN_COM_FCH_LFT_DRV : Bool;   // F505 Profinet network error furnace chamber lift drive
      PN_COM_TCH_TILT_DRV : Bool;   // F506 Profinet network error top chamber swivel drive
      PN_COM_TCH_LFT_DRV : Bool;   // F507 Profinet network error top chamber lift drive
      PN_COM_V7_LFT_DRV : Bool;   // F508 Profinet network error gate chamber valve lift drive
      PN_COM_V7_SW_DRV : Bool;   // F509 Profinet network error gate chamber valve swivel drive
      PN_COM_GCH_LFT_DRV : Bool;   // F510 Profinet network error gate chamber lift drive
      PN_COM_BEL_LFT_DRV : Bool;   // F511 Profinet network error bellow lift drive
      PN_COM_XT_HDL_SW_DRV : Bool;   // F512 Profinet network error crystal handling swivel drive
      PN_COM_XT_HDL_LFT_DRV : Bool;   // F513 Profinet network error crystal handling lift drive
      PN_COM_VALVE_BL_1 : Bool;   // F514 Profinet network error valve block level 1
      PN_COM_VALVE_BL_2 : Bool;   // F515 Profinet network error valve block level 2
      PN_COM_DEC_IO_K2 : Bool;   // F516 Profinet network error decentral IO-control Cabinet +K2
      PN_COM_DEC_IO_K5 : Bool;   // F517 Profinet network error decentral IO-control Cabinet +K5
      PN_COM_DEC_IO_K8 : Bool;   // F518 Profinet network error decentral IO-control Cabinet +K8
      PN_COM_DEC_IO_ACC : Bool;   // F519 Profinet network error decentral IO-control active cooling
      PN_COM_DEC_IO_FDR : Bool;   // F520 Profinet network error decentral IO-control feeder
      PN_COM_MAG : Bool;   // F521 Profinet network error decentral IO-control Magnet
      PN_COM_TEC_FLG_ENC : Bool;   // F522 Profinet network error technology flange lift encoder
      PN_COM_TEC_FLG_SW_ENC : Bool;   // F523 Profinet network error technology flange swivel encoder
      PN_COM_FCH_LFT_ENC : Bool;   // F524 Profinet network error furnace chamber lift encoder
      PN_COM_UP_FCH_SW_ENC : Bool;   // F525 Profinet network error upper furnace chamber swivel encoder
      PN_COM_LO_FCH_SW_ENC : Bool;   // F526 Profinet network error lower furnace chamber swivel encoder
      PN_COM_XT_HDL_SW_ENC : Bool;   // F527 Profinet network error crystal handling swivel encoder
      WTR_TMP_TEC_FLG : Bool;   // F528 water temp. technology flange
      WTR_FLW_TEC_FLG : Bool;   // F529 water flow technology flange
      WTR_TMP_GCH_ADDS : Bool;   // F530 water temp. gate chamber additions
      WTR_FLW_GCH_ADDS : Bool;   // F531 water flow gate chamber additions
      WTR_TMP_HLD_ACC : Bool;   // F532 water temp. holder active crystal cooling device
      WTR_FLW_HLD_ACC : Bool;   // F533 water flow holder active crystal cooling device
      BEL_LFT_ERR : Bool;   // F534 motor bellow lift error
      GCH_LFT_ERR : Bool;   // F535 motor gate chamber lift error
      V7_LFT_ERR : Bool;   // F536 motor gate chamber valve lift error
      V7_SW_ERR : Bool;   // F537 motor gate chamber valve swivel error
      TCH_LFT_ERR : Bool;   // F538 motor top chamber lift error
      TCH_TILT_ERR : Bool;   // F539 motor top chamber tilt error
      FCH_LFT_ERR : Bool;   // F540 motor furnace chamber lift error
      TEC_FLG_LFT_ERR : Bool;   // F541 motor technology flange lift error
      MAG_LFT_ERR : Bool;   // F542 motor magnet lift error
      XT_HDL_LFT_ERR : Bool;   // F543 motor crystal handling lift error
      XT_HDL_SW_ERR : Bool;   // F544 motor crystal handling swivel error
      XT_HDL_LFT_POS_REF : Bool;   // F545 crystal handling lift no reference
      XT_HDL_LFT_SLS : Bool;   // F546 safty limit switch crystal handling lift
      XT_HDL_SW_POS_REF : Bool;   // F547 crystal handling swivel no reference
      XT_HDL_SW_SLS : Bool;   // F548 safty limit switch crystal handling swivel
      COMP_ACC_AIR_PRS_LOW : Bool;   // F549 acc compressed air pressure is below limit
      COMP_SPL_AIR_PRS_LOW : Bool;   // F550 supply compressed air pressure is below limit
      EMS_HDL_DRV : Bool;   // F551 Emergency stop handling drives
      V2_11 : Bool;   // F552 vacuum valve V2.11 not open
      V3_3 : Bool;   // F553 vacuum valve V3.3 not open
      V3_4 : Bool;   // F554 vacuum valve V3.4 not open
      V22_1 : Bool;   // F555 vacuum valve V22.1 not open
      HTR1_COMM_ERR : Bool;   // F556 heater 1 communication error
      HTR2_COMM_ERR : Bool;   // F557 heater 2 communication error
      PWR_SPL_APF_ERR : Bool;   // F558 heater power supply APF error
      PWR_SPL_CTL_ERR : Bool;   // F559 heater power supply controller error
      HTR_1_ETH : Bool;   // F560 heater 1 earthing error
      HTR_2_ETH : Bool;   // F561 heater 2 earthing error
      HTR_ERH_COMM : Bool;   // F562 heater earthing communication error
      MAG_LFT_NOT_IN_POS : Bool;   // F563 magnet lifting unit not in highest position
      CR_ROT_TORQ_LIM : Bool;   // F564 crucible rotation drive exceeds torque limit
      FNC_OPN_DBL : Bool;   // F565 furnace opening is disabled - oxidation not completed
      MLT_GAP_NO_CONTACT : Bool;   // F566 no melt contact found within valid range
      HTR1_RCT_TMP : Bool;   // F567 Power supply heater 1 filter reactor temp. too high
      HTR2_RCT_TMP : Bool;   // F568 Power supply heater 2 filter reactor temp. too high
      ACC_24V_BUF_SPL : Bool;   // F569 ACC 24V DC buffer supply failure
      MAIN_24V_BUF_SPL : Bool;   // F570 Main 24V DC buffer supply failure
      WTR_TMP_VAC_BYP : Bool;   // F571 Water temperature vacuum bypass tube
      WTR_FLW_VAC_BYP : Bool;   // F572 Water flow vacuum bypass tube
      SEED_DET : Bool;   // F573 No seed detected within valid range
      SPARE_71_5 : Bool;   // F574
      SPARE_71_6 : Bool;   // F575
      SPARE_71_7 : Bool;   // F576
      SFT_HTR_SHUT_OFF : Bool;   // F577 Heater shut off due to safety matrix
      SFT_XT_ROT_OFF : Bool;   // F578 Crystal rotation shut off due to safety matrix
      SFT_CR_ROT_OFF : Bool;   // F579 Crucible rotation shut off due to safety matrix
      SFT_CR_LFT_DN : Bool;   // F580 Crucible lift down due to safety matrix
      WTR_FLW_CONE_WRN : Bool;   // F581 Cooling water flow cone warning
      WTR_TMP_CONE_WRN : Bool;   // F582 Cooling water temperature cone warning
      ABN_XT_WGT_CHG_RTE : Bool;   // F583 Abnormal crystal weight change rate
      ABN_XT_DIA_CHG_RTE : Bool;   // F584 Abnormal crystal diameter change rate
      HTR_1_SHRT_ABV_5_CNT : Bool;   // F585 Heater 1 short cuts detected above five counts
      HTR_1_SHRT_ABV_10_CNT : Bool;   // F586 Heater 1 short cuts detected above ten counts
      HTR_1_SHRT_ABV_20_CNT : Bool;   // F587 Heater 1 short cuts detected above twenty counts
      HTR_2_SHRT_ABV_5_CNT : Bool;   // F588 Heater 2 short cuts detected above five counts
      HTR_2_SHRT_ABV_10_CNT : Bool;   // F589 Heater 2 short cuts detected above ten counts
      HTR_2_SHRT_ABV_20_CNT : Bool;   // F590 Heater 2 short cuts detected above twenty counts
      SPARE_73_6 : Bool;   // F591
      SPARE_73_7 : Bool;   // F592
      SPARE : Array[74..127] of Byte;
   END_VAR
BEGIN
END_DATA_BLOCK

DATA_BLOCK "OP_MSG"   // DB143
{ S7_Optimized_Access := 'FALSE' }
VERSION : 0.0
// --------------------------------------------------------------------------------
//     program     :    OP_MSG
//     description :    Operator messages       
//     name        :    G. Eibelsh鋟ser
//     date        :    27.10.2007
// 
//     revision    :
//     name        :
//     date        :    
//                     (c)PVA TePla AG       
//     --------------------------------------------------------------------------------
   VAR
      BLANK : Int;   // msg:
      STEP_01 : Int := 1;   // msg: (do not change STEP_01...29)
      STEP_02 : Int := 2;   // msg:
      STEP_03 : Int := 3;   // msg:
      STEP_04 : Int := 4;   // msg:
      STEP_05 : Int := 5;   // msg:
      STEP_06 : Int := 6;   // msg:
      STEP_07 : Int := 7;   // msg:
      STEP_08 : Int := 8;   // msg:
      STEP_09 : Int := 9;   // msg:
      STEP_10 : Int := 10;   // msg:
      STEP_11 : Int := 11;   // msg:
      STEP_12 : Int := 12;   // msg:
      STEP_13 : Int := 13;   // msg:
      STEP_14 : Int := 14;   // msg:
      STEP_15 : Int := 15;   // msg:
      STEP_16 : Int := 16;   // msg:
      STEP_17 : Int := 17;   // msg:
      STEP_18 : Int := 18;   // msg:
      STEP_19 : Int := 19;   // msg:
      STEP_20 : Int := 20;   // msg:
      STEP_21 : Int := 21;   // msg:
      STEP_22 : Int := 22;   // msg:
      STEP_23 : Int := 23;   // msg:
      STEP_24 : Int := 24;   // msg:
      STEP_25 : Int := 25;   // msg:
      STEP_26 : Int := 26;   // msg:
      STEP_27 : Int := 27;   // msg:
      STEP_28 : Int := 28;   // msg:
      STEP_29 : Int := 29;   // msg:
      PD_10MBAR : Int := 30;   // msg:
      PD_1MBAR : Int := 31;   // msg:
      PD_01MBAR : Int := 32;   // msg:
      PD_005MBAR : Int := 33;   // msg:
      PD_FINAL : Int := 34;   // msg:
      PD_LEAK_TEST : Int := 35;   // msg:
      PD_CHECK_TIME : Int := 36;   // msg:
      PD_CHECK_LEAK_RATE : Int := 37;   // msg:
      DI_1_INIT_TIME : Int := 38;   // msg:
      DI_POWER_GAP1 : Int := 39;   // msg:
      DI_POWER_GAP2 : Int := 40;   // msg:
      DI_2_WAIT_TILL_CTL : Int := 41;   // msg:
      DI_3_MELT_TEMP_CTL : Int := 42;   // msg:
      DI_4_SEED_DOWN : Int := 43;   // msg:
      DI_5_SEED_INTO_MELT : Int := 44;   // msg:
      DI_6_WAIT_TIME1 : Int := 45;   // msg:
      DI_7_WAIT_TIME2 : Int := 46;   // msg:
      DI_8_TEMP_GAP : Int := 47;   // msg:
      WAIT_FOR_AUTO : Int := 48;   // msg:
      OPEN_GATE_VALVE : Int := 49;   // msg:
      NE_DIA_REDUCTION1 : Int := 50;   // msg:
      NE_DIA_REDUCTION2 : Int := 51;   // msg:
      NE_DIA_CONSTANT : Int := 52;   // msg:
      SH_TEMP_GAP : Int := 53;   // msg:
      SH_WAIT_TILL_GROWTH_CTL : Int := 54;   // msg:
      SH_WITH_GROWTH_CTL : Int := 55;   // msg:
      SH_TRANSITION_TO_BODY : Int := 56;   // msg:
      BY_WAIT_TILL_DIA_CTL : Int := 57;   // msg:
      SD_WAIT_TILL_VENTING : Int := 58;   // msg:
      SD_WAIT_TILL_LEAK_TEST : Int := 59;   // msg:
      SD_VENTING : Int := 60;   // msg:
      CLOSE_GATE_VALVE : Int := 61;   // msg:
      VENTING_GATE : Int := 62;   // msg:
      PUMP_DOWN_GATE : Int := 63;   // msg:
      RE_CRYSTAL_UP : Int := 64;   // msg:
      RE_CRYSTAL_TO_POS : Int := 65;   // msg:
      RE_CRUCIBLE_TO_POS : Int := 66;   // msg:
      RE_WAIT_TILL_XT_COOL : Int := 67;   // msg:
      RE_REMOVE_CRYSTAL : Int := 68;   // msg:
      RE_WAIT_FOR_DIP : Int := 69;   // msg:
      OP_CALL_ALM : Int := 70;   // msg:
      PD_WAIT_DRV_CAL : Int := 71;   // msg:
      DI_AUTO_THR_ADJ : Int := 72;   // msg:
      BY2_RAMP_ACTIVE : Int := 73;   // msg:
      EMG_ACTIVE : Int := 74;   // msg:
      FDR_IS_MOVING_TO_HOME : Int := 75;   // msg:
      CONNECT_HOPPER : Int := 76;   // msg:
      ME_CHECK_LRT_FDR : Int := 77;   // msg:
      MOVE_FDR_TO_HOME : Int := 78;   // msg:
      PD_PRG_PRS : Int := 79;   // msg: Abpumpen
      PD_PRG : Int := 80;   // msg: Sp黮en
      PD_WAIT_TME : Int := 81;   // msg: Wartezeit vor Lecktest
      PD_WAIT_TME_V2 : Int := 82;   // msg: Wartezeit f黵 Freigabe V2
      PD_CHECK_PLANT : Int := 83;   // msg: Enddruck nicht erreicht - Anlage 黚erpr黤en
      PD_INI_PRS_NOT_RCH : Int := 84;   // msg: Anfangsdruck nicht erreicht - Anlage 黚erpr黤en
      SD_CHECK_LEAK_RATE : Int := 85;   // msg: Leckrate pr黤en
      ME_CHK_DST_MLT_TO_FNL : Int := 86;   // msg: Abstand Schmelze - Trichter pr黤en
      DI_RMLT_PRV_NE : Int := 87;   // msg: Vorherigen Hals r點kschmelzen - Remelting of previous neck
      RE_HTR_TMP_RSD : Int := 88;   // msg: Heizer Temperatur wird angehoben - Heater temperature is raised
      RE_CR_LWD : Int := 89;   // msg: Tiegel wird abgesenkt - Crucible is lowered
      SD_WAIT_UNTIL_COOL_DN : Int := 90;   // msg: Temperatur zu hoch zum Fluten - Temperatur too high for venting
      SD_WAIT_AFT_VENT : Int := 91;   // msg: Wartezeit nach dem Bel黤ten - Wait time after venting
      SD_FIL_FSH_ACTIVE : Int := 92;   // msg: Filterreinigung ist aktiv - Filter regeneration is active
      RE_HTR_PWR_RSD : Int := 93;   // msg: Heizer Leistung wird angehoben - Heater power is raised
      DI_8_PWR_GAP : Int := 94;   // msg: Schritt 8: Leistungssprung - Step 8: Power gap
      SPARE_095 : Int := 95;   // msg:
      SPARE_096 : Int := 96;   // msg:
      SPARE_097 : Int := 97;   // msg:
      MOB_FDR_DOCK : Int := 98;   // yes: Bitte mobiler Feeder andocken!
      MOB_FDR_UNDOCK : Int := 99;   // yes: Bitte mobiler Feeder abdocken!
      MOB_FDR_TUBE_IN : Int := 100;   // yes: Bitte mobiler Feeder Rohr einfahren!
      START_NEW_INGOT : Int := 101;   // yes/no: Soll ein neuer Ingot gezogen werden?
      MOB_FDR_TUBE_DRV_IN : Int := 102;   // msg: Mobiler Feeder; Rohr wird eingefahren
      MOB_FDR_TUBE_DRV_OUT : Int := 103;   // msg: Mobiler Feeder; Rohr wird ausgefahren
      MOB_FDR_FEED_SEQ_RUN : Int := 104;   // msg: Mobiler Feeder; Feeding Sequenz aktiv
      RE_SEQ_FINISH : Int := 105;   // msg: Entnahme Sequenz beendet
      SPARE_106 : Int := 106;   // msg:
      SPARE_107 : Int := 107;   // msg:
      SPARE_108 : Int := 108;   // msg:
      SPARE_109 : Int := 109;   // msg:
      STEP_30 : Int := 110;   // msg:
   END_VAR
BEGIN
END_DATA_BLOCK

DATA_BLOCK "CNF"   // DB144
{ S7_Optimized_Access := 'FALSE' }
VERSION : 0.0
// --------------------------------------------------------------------------------
//     program     :    CNF
//     description :    configuration data
// 
//     name        :
//     date        :
// 
//                     (c) PVA CGS GmbH
//     --------------------------------------------------------------------------------
//     CONF_xxx                0   device not installed
//                             1   device installed
// 
//     info        :    trigger mode:  #0= Trigger 黚er Break-Out Box (digital)
//                                     #1= Trigger 黚er TCP-Kommando
//     
// 
//     EKZ hardware device configuration:
//     
//     Bit  0  :   crystal lift
//     Bit  1  :   crystal rotation
//     Bit  2  :   crucible lift
//     Bit  3  :   crucible rotation
//     Bit  4  :   temperature control heater 1
//     Bit  5  :   heater 2 (bottom)
//     Bit  6  :   Ar MFC 1
//     Bit  7  :   Ar MFC 2
//     Bit  8  :   Camera (single camera mode)
//     Bit  9  :   not used
//     Bit 10  :   Magnet resistive
//     Bit 11  :   Magnet superconductive
//     Bit 12  :   Feeder (old design)
//     Bit 13  :   Pressure control valve
//     Bit 14  :   Cooling water
//     Bit 15  :   crystal load cell
//     Bit 16  :   melt level laser measurement system
//     Bit 17  :   crystal drop out protection
//     Bit 18  :   melt contact control 
//     Bit 19  :   Camera (stereo camera mode)
//     Bit 20  :   pressure gauge gate chamber
//     Bit 21  :   shoulder diameter control
//     Bit 22  :   screw pump reset
//     Bit 23  :   gate chamber lift encoder 
//     Bit 24  :   power supply reset
//     Bit 25  :   active crystal cooling device
//     Bit 26  :   Mobile Feeder
//     Bit 27  :   Stationary Feeder (new design 2012)
//     Bit 28  :   power control heater 1
//     Bit 29  :   SiO Bypass with cooling tube without filter
//     Bit 30  :   Gap Controller
//     Bit 31  :   SiO Bypass filter with cleaning of main filter during process
//     
//     
//     ACT_DVC_CNF :   DWORD   :=   2#0110_0011_0001_1110_0110_1000_1111_1111   
//                             :=  16#631E68FF
//     ---------------------------------------------------
   VAR
      ACT_DVC_CNF : DWord := DWORD#16#631E_68FF;   // actual device configuration - see legend above
      CONF_PWR_SPL_TYPE : Int := 1;   // power supply type- 1: TLU, 2: INJET
      CONF_WTR_SPL_TYPE : Int := 2;   // cooling water supply type: 1 - EKZ 2700; 2 - EKZ 3500
      CONF_GTE_CBR_DOOR : Bool := TRUE;   // gate chamber with door : 1, gate tube without door: 0
      CONF_CGT_BAR_1000 : Bool := TRUE;   // 1000 mbar Baratron gate chamber
      CONF_CLF_BAR_1000 : Bool := TRUE;   // 1000 mbar Baratron furnace chamber
      CONF_VALVE_POS_DET : Bool := TRUE;   // position detection for vacuum valves
      CONF_BREAKER_FLT_DET : Bool := TRUE;   // inputs for aux contacts of circuit breaker
      CONF_PRS_CTL_ANA : Bool := TRUE;   // pressure control valve with analog setpoint input
      CONF_DRV_EKZ2700 : Bool;   // drive configuration EKZ 2700
      CONF_DRV_CAL : Bool;   // drive calibration (old EKZ 2700)
      CONF_DRV_WHILE_LRT : Bool;   // drives active when leakrate is calculated
      CONF_MAG_LFT : Bool := TRUE;   // magnet lifting device installed
      CONF_DP_DIAG_ON : Bool := TRUE;   // dp diagnosis function active
      CONF_SH_PAR_FNCT : Bool := TRUE;   // function type for shoulder parameters: 0= diameter, 1= length
      CONF_HND_HYD : Bool;   // hydraulic handling of furnace and gate chamber with software control
      CONF_FDR : Bool;   // granular feeder installed (old design)
      CONF_LSR_LVL : Bool;   // laser device for melt level detection installed
      CONF_AR_V_16 : Bool;   // Argon upstream valve(s) V16.x present
      CONF_VAC_V2_2 : Bool;   // Vacuum valve V2.2 present
      CONF_DIFF_PRS : Bool;   // differential pressure switch in vacuum line installed
      CONF_ENC_TYPE : Bool := TRUE;   // 1:= absolute encoders, 0:= incremental encoders
      CONF_ENC_HNDL : Bool := TRUE;   // 1:= encoder for handling lift is installed, 0:= not installed
      CONF_PWR_SPL_L2 : Bool := TRUE;   // power supplies with profibus interface
      CONF_MFC_L2 : Bool := TRUE;   // MFC with profibus interface
      CONF_CAM_2 : Bool;   // camera 2 installed
      CONF_LOAD_CELL : Bool;   // 1:= crystal load cell is installed, 0:= not installed
      CONF_24V_UPS : Bool := TRUE;   // 1:= 24V UPS installed, 0:= not installed
      VOLUME_LEAK_TEST : Real := 3000.0;   // volume used for leak test [l]
      VOLUME_MAIN_FIL : Real := 600.0;   // volume of main filter used for leak test [l]
      VOLUME_BYP_FIL : Real := 600.0;   // volume of bypass filter used for leak test [l]
      VOLUME_MOB_FDR : Real := 250.0;   // volume of mobile feeder used for leak test [l]
      WTR_TMP_WRN : Real := 50.0;   // water temperature limit for warning
      MAX_WTR_TMP_LIM : Real := 65.0;   // water temperature limit for shut down of heater
      MIN_WTR_FLW_COOL_FLG : Real := 5.0;   // minimum water flow limit cooling flange vacuum pipe
      MIN_WTR_FLW_XT_SFT : Real := 5.5;   // minimum water flow limit seed shaft
      MIN_WTR_FLW_GCH : Real := 15.0;   // minimum water flow limit gate chamber
      MIN_WTR_FLW_GCH_H : Real := 7.5;   // minimum water flow limit gate chamber valve housing
      MIN_WTR_FLW_GCH_V : Real := 5.5;   // minimum water flow limit gate chamber valve
      MIN_WTR_FLW_VPTS : Real := 3.0;   // minimum water flow limit view ports
      MIN_WTR_FLW_TCH : Real := 15.0;   // minimum water flow limit top chamber
      MIN_WTR_FLW_TEC_CHB : Real := 8.0;   // minimum water flow limit technology chamber
      MIN_WTR_FLW_FCH : Real := 15.0;   // minimum water flow limit furnace chamber
      MIN_WTR_FLW_VSL : Real := 8.0;   // minimum water flow bottom chamber
      MIN_WTR_FLW_SOC_BCH : Real := 5.5;   // minimum water flow limit socket bottom chamber
      MIN_WTR_FLW_CUR_FEED : Real := 5.5;   // minimum water flow limit current feed throughs F
      MIN_WTR_FLW_CFT_2 : Real := 5.5;   // minimum water flow limit current feed throughs B
      MIN_WTR_FLW_PWR_CAB : Real := 7.5;   // minimum water flow limit high current cables
      MIN_WTR_FLW_CR_SFT : Real := 7.5;   // minimum water flow limit crucible shaft
      MIN_WTR_FLW_CR_SFT_F : Real := 5.0;   // minimum water flow limit crucible shaft F
      MIN_WTR_FLW_CR_SFT_B : Real := 5.0;   // minimum water flow limit crucible shaft B
      MIN_WTR_FLW_PWR_HTR_1 : Real := 30.0;   // minimum water flow limit heater power supply
      MIN_WTR_FLW_INJ_HTR_1 : Real := 50.0;   // minimum water flow limit Injet heater power supply
      MIN_WTR_FLW_ACC_IN : Real := 5.0;   // minimum water flow limit active cooling
      MIN_WTR_FLW_GCH_ADDS : Real := 2.5;   // minimum water flow limit chamber parts, view ports
      MIN_WTR_FLW_PU : Real := 5.0;   // minimum water flow limit pump unit
      MIN_WTR_FLW_MAG_COMP : Real := 4.0;   // minimum water flow limit magnet compressor unit 4
      MIN_WTR_FLW_MAG_CAB : Real := 8.0;   // minimum water flow LIMIT magnet power supply
      MIN_WTR_FLW_VAC_BYP : Real := 10.0;   // minimum water flow limit vacuum bypass tube image acquisition
      IMG_AQI_TRG : Int := 500;   // trigger time in [ms]
      CP_LADDR : Word := WORD#16#0190;   // add: 400
      CAM_1_CON_ID_SEND : Int := 1;
      CAM_1_CON_ID_RECV : Int := 2;
      CAM_2_CON_ID_SEND : Int := 3;
      CAM_2_CON_ID_RECV : Int := 4;
      CNF_XT_POS : Struct
         d0 : Real := 1.0;   // distance for switching to red. speed
         td : Real := 0.1;   // delay time
         t_ramp : Real := 8.0;   // time to reduce speed from v_max to 0
         v_max : Real := 1000.0;   // max speed in fast mode
         v_low : Real := 1.0;   // min value for reduced speed
      END_STRUCT;
      CNF_CR_POS : Struct
         d0 : Real := 0.5;   // distance for switching to red. speed
         td : Real := 0.5;   // delay time
         t_ramp : Real := 4.0;   // time to reduce speed from v_max to 0
         v_max : Real := 260.0;   // max speed in fast mode
         v_low : Real := 1.0;   // min value for reduced speed
      END_STRUCT;
      DIP_XT_POS : Real := 3300.0;   // crystal position in dipping must be below this value
      DIP_XT_SPD_UP : Real := 300.0;   // crystal speed for moving up in dipping mode
      NECK_SLOPE_1 : Real := 0.5;   // [mm/min] diameter reduction neck
      NECK_SLOPE_2 : Real := 0.25;   // [mm/min] diameter reduction neck
      NECK_DELTA_SLOPE_1 : Real := 1.5;   // [mm] final dia + delta = end dia 1
      RE_RMP_RTE_HTR : Real := 8.0;   // ramp rate htr[癈/min]
      RE_RMP_RTE_XT_ROT : Real := 1.0;   // ramp rate crystal rotation [rpm/min]
      RE_RMP_RTE_CR_ROT : Real := 4.0;   // ramp rate crucible rotation [rpm/min]
      RE_XT_SPD_FST : Real := 100.0;   // fast speed for xtal removal [mm/min]
      RE_CR_SPD : Real := 2.0;   // speed for crucible [mm/min]
      RE_PRS_DIFF : Real := 5.0;   // pressure difference for open gate [mbar]
      XT_LFT_SPEED_NORM : Real := 8.0;   // [mm/min] normal xtal lift speed
      XT_LFT_SPEED_FAST : Real := 500.0;   // [mm/min] fast xtal lift speed
      XT_LO_POS : Real := 2500.0;   // [mm] lowest position for moving down xtal lift while gate valve closed
      XT_CAL_POS : Real := 200.0;   // [mm] start position for xtal lift calibration
      CR_CAL_POS : Real := 5.0;   // [mm] start position for cruc lift calibration
      XT_LFT_SPD_DRV_CAL : Real := 0.8;   // [mm/min] xtal lift speed for drive calibration
      XT_ROT_DRV_CAL : Real := 0.9;   // [rpm] xtal rotation for drive calibration
      XT_SPD_WHILE_LRT : Real := 1.0;   // [mm/min] xtal lift speed when leakrate is calculated
      XT_ROT_WHILE_LRT : Real := 8.0;   // [rpm] xtal rotation when leakrate is calculated
      CRUC_LFT_SPEED_NORM : Real := 0.5;   // [mm/min] normal crucible lift speed
      CRUC_LFT_SPEED_FAST : Real := 50.0;   // [mm/min] fast crucible lift speed
      CR_LFT_SPD_DRV_CAL : Real := 0.05;   // [mm/min] cruc lift speed for drive calibration
      CR_ROT_DRV_CAL : Real := 0.5;   // [rpm] cruc rotation for drive calibration
      CR_SPD_WHILE_LRT : Real := 0.1;   // [mm/min] cruc lift speed when leakrate is calculated
      CR_ROT_WHILE_LRT : Real := 2.0;   // [rpm] cruc rotation when leakrate is calculated
      CR_SPD_LSR_ME_DET : Real := 2.0;   // [mm/min] cruc lift speed for melt level detection with laser device
      LSR_LVL_RANGE : Real := 10.0;   // range for melt level laser detection system in [mm]
      XT_DIA_RANGE : Real := 500.0;   // range for xtal diameter [mm]
      XT_LFT_RANGE : Real := 10.0;   // range for xtal lift [mm/min]
      XT_ROT_RANGE : Real := 20.0;   // range for xtal rotation [RPM]
      CR_LFT_RANGE : Real := 2.6;   // range for crucible lift [mm/min]
      CR_ROT_RANGE : Real := 20.0;   // range for crucible rotation [RPM]
      HTR_1_PWR_RANGE : Real := 216.0;   // range for heater 1 power [kW]
      HTR_1_CUR_RANGE : Real := 3600.0;   // range for heater 1 current [A]
      HTR_1_VLT_RANGE : Real := 60.0;   // range for heater 1 voltage [V]
      HTR_1_RES_RANGE : Real := 50.0;   // range for heater 1 resistance [mOhm]
      HTR_1_TMP_RANGE_LOW : Real := 300.0;   // range for heater 1 temperature [癈] low value
      HTR_1_TMP_RANGE_HI : Real := 2000.0;   // range for heater 1 temperature [癈] high value
      HTR_2_PWR_RANGE : Real := 130.0;   // range for heater 2 power [kW]
      HTR_2_CUR_RANGE : Real := 2600.0;   // range for heater 2 current [A]
      HTR_2_VLT_RANGE : Real := 50.0;   // range for heater 2 voltage [V]
      HTR_2_RES_RANGE : Real := 50.0;   // range for heater 2 resistance [mOhm]
      HTR_2_TMP_RANGE_LOW : Real;   // range for heater 2 temperature [癈] low value
      HTR_2_TMP_RANGE_HI : Real;   // range for heater 2 temperature [癈] high value
      MAG_1_PWR_RANGE : Real;   // range for magnet coil 1 power [kW]
      MAG_1_CUR_RANGE : Real := 150.0;   // range for magnet coil 1 current [A]
      MAG_1_VLT_RANGE : Real;   // range for magnet coil 1 voltage [V]
      MAG_2_PWR_RANGE : Real;   // range for magnet coil 2 power [kW]
      MAG_2_CUR_RANGE : Real := 150.0;   // range for magnet coil 2 current [A]
      MAG_2_VLT_RANGE : Real;   // range for magnet coil 2 voltage [V]
      SET_MAG_RMP_RTE : Real := 3.132;   // ramp rate of magnet current set point in [A/min]
      MAG_WORK_POS : Real := 800.0;   // range working position release magnet power
      MLT_TMP_1_RANGE_LOW : Real := 900.0;   // range for melt 1 temperature [癈] low value
      MLT_TMP_1_RANGE_HI : Real := 1600.0;   // range for melt 1 temperature [癈] high value
      GAS_FLW_1_RANGE : Real := 200.0;   // range of MFC 1
      GAS_FLW_2_RANGE : Real := 50.0;   // range of MFC 2
      CLF_PRS_RANGE : Real := 1000.0;   // range for pressure in lower furnace chamber [mBar]
      CAM_PIX_FULL_LINE : Real := 1376.0;   // amount of pixel in a full line in the specified window (measured)
      SET_HND_LFT_SPD : Real := 50.0;   // gate lift speed setpoint
      SET_HND_SWL_SPD : Real := 20.0;   // gate swivel speed setpoint
      MAX_DIFF_PRS_FDR_FNC : Real := 25.0;   // max.difference prs fnc - prs fdr for V11 to open [mbar]
      FDR_VOL_LEAK_TEST : Real := 126.0;   // feeder volume used for leak test [l]
      FDR_PRS_V11_TST : Real := 50.0;   // pressure for final V11 test after feeding sequence [mbar]
      FDR_PUR_PRS_HI : Real := 700.0;   // NOT USED! high pressure limit feeder pump and purge cycle [mbar]
      FDR_PUR_PRS_LO : Real := 50.0;   // low pressure limit feeder pump and purge cycle [mbar]
      MAX_FDR_TUBE_MVE_TME : Int := 45;   // max. time for feeder tube movement
      FDR_PMP_DN_TME : Int := 20;   // pump down time for feeder housing after cover is closed in [min]
      HYD_PMP_DLY : Int := 20;   // delay time in 100ms for hydraulic pump to build up pressure
      SEED_TMP_CTL_POS_LIM : Real := 2000.0;   // position limit for definition of "seed hot" (manual mode)
      SEED_TMP_CTL_HI_POS : Real := 400.0;   // stop position for hot seed in manual mode
      XT_LD_MAX : Real := 700.0;   // maximum weight of crystal load cells
      XT_LFT_REF_VAL : Real := 23629.0;   // reference position of crystal lift encoder =>> 70.0 mm
      CR_LFT_REF_VAL : Real := 90112.0;   // reference position of crucible lift encoder =>> 10.0 mm
      HDL_LFT_REF_VAL : Real := 40960.0;   // reference position of handling lift encoder =>> 0.0 mm
      XT_WGT_RTE_ORD : Real := 600.0;   // time between two values used for calculation of first derivative
      RHO_SOL_SI_ROOM : Real := 2.33E-06;   // density of solid Si at room temperature [kg/mm^3]
      RHO_SOL_SI_MLT : Real := 2.28E-06;   // density of solid Si near melt temperature [kg/mm^3]
      RHO_LI_SI : Real := 2.55E-06;   // density of liquid Si [kg/mm^3]
      PI : Real := 3.141593;   // Zahl PI
      RST_LIM_XT_ORB_NE : Real := 1.0;   // reset limit crystal orbiting in neck phase in [mm]
      RST_LIM_XT_ORB_SH : Real := 1.0;   // reset limit crystal orbiting in shoulder phase in [mm]
      RST_LIM_XT_ORB_BY : Real := 1.0;   // reset limit crystal orbiting in body phase in [mm]
      CTL_MLT_DRIFT_TF : Real := 30.0;   // sec
      MAX_VALID_DRIFT_RTE : Real := 1.0;   // mm/min
      CR_SPD_COF_RANGE : Real := 200.0;   // range for crucible speed coeffizeint range [%]
      SPD_CALC_AT_BY_LEN : Real;   // start body length FOR calculation OF effective speed [mm]
      RM_MLT_AFT_PRC : Real := 5.0;   // target amount OF remaining melt after process (only used FOR length calculati
      TMP_LIM_VENTING : Real := 1000.0;   // heater temperature must be below this value for venting the furnace
      XT_HDL_SW_ENC_RATIO : Real := 360.0;   // 360?1 gear ratio encoder crystal handling swivel drive
      FCH_ENC_RATIO : Real := 12.0;   // 12:1 gear ratio encoder furnace chamber lift drive
      TEC_FLG_ENC_RATIO : Real := 8.0;   // 8:1 gear ratio encoder technology flange lift drive
      LO_FCH_SW_ENC_RATIO : Real := 38.57144;   // 504:54 gear ratio encoder lower furnace chamber swivel = 360*54/504
      UP_FCH_SW_ENC_RATIO : Real := 38.57144;   // 504:54 gear ratio encoder upper furnace chamber swivel
      TEC_FLG_SW_ENC_RATIO : Real := 38.57144;   // 504:54 gear ratio encoder technolegy flange swivel
      XT_HDL_SW_REF_POS : Real := 143.0;   // Referenz postion encoder crystal handling swivel drive
      TEC_FLG_REF_POS : Real := 20.0;   // Referenz postion encoder technology flange lift drive
      FCH_REF_POS : Real := 20.0;   // Referenz postion encoder furnace chamber lift drive
      LO_FCH_SW_REF_POS : Real := 90.009;   // Referenz postion encoder lower furnace chamber swivel
      UP_FCH_SW_REF_POS : Real := 90.009;   // Referenz postion encoder upper furnace chamber swivel
      TEC_FLG_SW_REF_POS : Real := 90.009;   // -------------------------------------------------
      d : Real := 150.0831;   // 150.0 - diameter winding drum
      cpr_xt : Real := 4096.0;   // no of counts
      cpr : Real := 4096.0;   // no of counts
      P_CR : Real := 5.0;   // pitch spindle crucible lift
      P_HND : Real := 10.0;   // pitch spindle handling lift --------Process Antrieb Position limit switch
      xt_high_pos : Real := 100.0;   // 325.0 crystal upper position absolute
      xt_low_pos : Real := 4500.0;   // 4500.0 crystal lower position absolute
      xt_lft_rmp : Real := 50.0;   // crystal lift ramp (upper and lower)
      cr_high_pos : Real := 940.0;   // 940.0 crucible upper position opened plant (vorher 600.0)
      cr_low_pos : Real := 0.5;   // 10.0 crucible lower position absolute
      cr_lft_rmp : Real := 15.0;   // crucible lift ramp (upper and lower)
      MOB_FDR_TUBE_SPD_INC : Int := 1;   // mobile feeder tube speed increment in [%]
      MOB_FDR_TUBE_SPD : Int := 50;   // mobile feeder tube speed in [0..100%]
      MOB_FDR_PRS_INC : Real := 30.0;   // prs. inc. while doing pressure drop test in undock sequence in [mbar]
      hnd_high_pos : Real := 1110.0;   // handling upper position
      hnd_low_pos : Real;   // handling lower position
      hnd_low_pos_clf : Real := 350.0;   // hnd lowest pos if CLF not in pulling position
      hnd_low_pos_cgt : Real;   // hnd lowest pos if CGT not in pulling position (mit AKK, vorher 150.0)
      hnd_lft_rmp : Real := 40.0;   // handling lift ramp (upper and lower)
      swl_enb_CUF : Real := 600.0;   // lowest position for handling swivel with CUF
      swl_enb_CGT : Real := 300.0;   // lowest position for handling swivel without CUF
      V9_close_pos : Real := 20.0;   // for close request V9
      stop_up : Real := 200.0;   // stop to secure crystal with safty fork
      stop_dn : Real := 1000.0;   // stop in outer pos. to remove crystal
      Pos_Offset : Real := -100.0;   // offset to avoid position 0 (bus-error-detect)
      max_count : Int := 50;   // maximum number of cycles
      ACC_FNC_PRS_LIM : Real := 950.0;   // furnace pressure limit for closing gas inlet valves (V4 + V5 + V6) while ventin
      ACC_SET_GAS_1_FLW_VNT : Real := 20.0;   // gas flow set point while venting furnace through valve V5
      TEC_FLG_MAX_POS : Real := 910.0;   // technology flange lift up max to 900 mm
      TEC_FLG_REL_DRV_POS : Real := 40.0;   // technology flange lift position release furnace chamber lift
      TEC_FLG_REL_SW_POS : Real := 750.0;   // technology flange lift position release swivel flange with active cooling devi
      TEC_FLG_SW_HOME_POS : Real;   // technology flange limit switch swiveling home position (in)
      TEC_FLG_SW_CLN_POS : Real := 120.0;   // technology flange limit switch swiveling cleaning position
      TEC_FLG_SW_MAX_POS : Real := 167.0;   // technology flange limit switch swiveling max.position (out)
      FCH_LFT_MAX_POS : Real := 1170.0;   // furnace chamber lift max. upper position
      FCH_REL_SW_POS : Real := 200.0;   // furnace chamber lift position release swivel out
      UP_FCH_SW_HOME_POS : Real;   // upper furnace chamber limit switch swiveling home position (in)
      UP_FCH_SW_CLN_POS : Real := 120.0;   // upper furnace chamber limit switch swiveling cleaning position
      UP_FCH_SW_MAX_POS : Real := 167.0;   // upper furnace chamber limit switch swiveling max. position (out)
      LO_FCH_SW_HOME_POS : Real;   // lower furnace chamber limit switch swiveling home position (in)
      LO_FCH_SW_PARK_POS : Real := 90.0;   // lower furnace chamber limit switch swiveling park position
      LO_FCH_SW_CLN_POS : Real := 120.0;   // lower furnace chamber limit switch swiveling cleaning position
      LO_FCH_SW_MAX_POS : Real := 150.0;   // lower furnace chamber limit switch swiveling max. position (out)
      XT_HDL_MAX_UP_POS : Real := 2200.0;   // cystal handling max. lifting up position
      XT_HDL_SW_OUT_POS : Real := 10.0;   // crystal handling max. swiveling position (out)
      XT_HDL_SW_OUT_DN_POS : Real := 100.0;   // cystal handling lifting down limit by swivel out position
      XT_HDL_TRP_DN_POS : Real := 300.0;   // cystal handling lifting down limit by transport cart's position
      XT_HDL_SW_IN_DN_POS : Real := 1000.0;   // cystal handling lifting down limit by swivel in position
      XT_HDL_SW_IN_UP_POS : Real := 1600.0;   // cystal handling lifting up limit by swivel in position
      XT_HDL_MAX_DN_POS : Real := 10.0;   // cystal handling max. lifting down position
      XT_HDL_LFT_TRP_POS : Real := 135.0;   // cystal handling lifting transport cart's position
      XT_HDL_SW_IN_TRP_POS : Real := 53.0;   // cystal handling swiveling transport cart's position
      XT_ACP_LFT_MID_POS : Real := 1500.0;   // cystal acceptance lifting middle position
      XT_ACP_LFT_LWR_POS : Real := 1480.0;   // cystal acceptance lifting lower position
      XT_HDL_SW_IN_POS : Real := 143.0;   // cystal acceptance swiveling position 143?in)
      XT_ACP_LFT_UPR_POS : Real := 1550.0;   // cystal acceptance lifting upper position
      XT_CLP_LDC_CAL : Real := 1.313768;   // cystal handling calibration factor loading cell
      REL_V21_POS_V1 : Real := 10.0;   // Release V21 "Oxidation valve" by open angle of throttle valve V1
      XT_HDL_SW_IN_CRU_POS : Real := 181.0;   // Crucible swiveling position 181?in)
      XT_HDL_LFT_CRU_UP_POS : Real := 1490.0;   // XT-Lift max upper pos at swiveling at Crucible
      XT_HDL_LFT_REL_SW_IN : Real := 840.0;   // XT-Lift max upper pos at swiveling at Crucible
      S_CAM_ANG_BETA : Real := 4.0;   // angle difference between two cameras, gemessen im CAD f黵 CGS1218
      MAX_GAP_OFFS : Real := 10.0;   // maximum melt gap offset in [mm]
      AVG_GAP_OFFS_TMP_RNG : Real := 10.0;   // max. temperature increment range of average gap offset controller in [癈]
      AVG_GAP_OFFS_PWR_RNG : Real := 5.0;   // max. power increment range of average gap offset controller in [KW]
      TEC_FLG_OP_BRK_POS : Real := 100.0;   // tech. flange operater unlock position during lifting down [mm]
      UP_FCH_OP_BRK_POS : Real := 70.0;   // upper furnace operater unlock position during lifting down [mm] (#128: 50mm,
      LO_FCH_OP_BRK_POS : Real := 175.0;   // lower furnace operater unlock position during lifting down [mm] (#128: 165mm,
      V22_OP_TME : Int := 3000;   // duration V22 opened for blowback pulse of SiO filter [ms]
      AMT_OF_V22_BB : Int := 1;   // amount of filter blow backs through V22
      MAX_PRS_AR_VSL : Real := 2.2;   // max. pressure argon vessel in [bar_abs]
      MIN_PRS_AR_VSL : Real := 1.1;   // min. pressure argon vessel in [bar_abs]
   END_VAR
BEGIN
END_DATA_BLOCK

DATA_BLOCK "SM_FLT_ACKN"   // DB145
{ S7_Optimized_Access := 'FALSE' }
VERSION : 0.0
// --------------------------------------------------------------------------------
//     program     :    SM_FLT_ACKN
//     description :    List of acknowledged fault signals      
//     name        :    G. Eibelsh鋟ser
//     date        :    01.12.99
// 
//     revision    :    Anzahl der Alarmworte verdoppelt
//     name        :    G. Eibelsh鋟ser
//     date        :    04.01.2007
// 
//                     (c)PVA TePla AG         
//     --------------------------------------------------------------------------------
   VAR
      ALARM_WORD_0 : Word;   // F001 - F016
      ALARM_WORD_1 : Word;   // F017 - F032
      ALARM_WORD_2 : Word;   // F033 - F048
      ALARM_WORD_3 : Word;   // F049 - F064
      ALARM_WORD_4 : Word;   // F065 - F080
      ALARM_WORD_5 : Word;   // F081 - F096
      ALARM_WORD_6 : Word;   // F097 - F112
      ALARM_WORD_7 : Word;   // F113 - F128
      ALARM_WORD_8 : Word;   // F129 - F144
      ALARM_WORD_9 : Word;   // F145 - F160
      ALARM_WORD_10 : Word;   // F161 - F176
      ALARM_WORD_11 : Word;   // F177 - F192
      ALARM_WORD_12 : Word;   // F193 - F208
      ALARM_WORD_13 : Word;   // F209 - F224
      ALARM_WORD_14 : Word;   // F225 - F240
      ALARM_WORD_15 : Word;   // F241 - F256
      ALARM_WORD_16 : Word;   // F257 - F272
      ALARM_WORD_17 : Word;   // F273 - F288
      ALARM_WORD_18 : Word;   // F289 - F304
      ALARM_WORD_19 : Word;   // F305 - F320
      ALARM_WORD_20 : Word;   // F321 - F336
      ALARM_WORD_21 : Word;   // F337 - F352
      ALARM_WORD_22 : Word;   // F353 - F368
      ALARM_WORD_23 : Word;   // F369 - F384
      ALARM_WORD_24 : Word;   // F385 - F400
      ALARM_WORD_25 : Word;   // F401 - F416
      ALARM_WORD_26 : Word;   // F417 - F432
      ALARM_WORD_27 : Word;   // F433 - F448
      ALARM_WORD_28 : Word;   // F449 - F464
      ALARM_WORD_29 : Word;   // F465 - F480
      ALARM_WORD_30 : Word;   // F481 - F496
      ALARM_WORD_31 : Word;   // F497 - F512
      ALARM_WORD_32 : Word;   // F513 - F528
      ALARM_WORD_33 : Word;   // F529 - F544
      ALARM_WORD_34 : Word;   // F545 - F560
      ALARM_WORD_35 : Word;   // F561 - F576
      ALARM_WORD_36 : Word;   // F577 - F592
      ALARM_WORD_37 : Word;   // F593 - F608
      ALARM_WORD_38 : Word;   // F609 - F624
      ALARM_WORD_39 : Word;   // F625 - F640
      ALARM_WORD_40 : Word;   // F641 - F656
      ALARM_WORD_41 : Word;   // F657 - F672
      ALARM_WORD_42 : Word;   // F673 - F688
      ALARM_WORD_43 : Word;   // F689 - F704
      ALARM_WORD_44 : Word;   // F705 - F720
      ALARM_WORD_45 : Word;   // F721 - F736
      ALARM_WORD_46 : Word;   // F737 - F752
      ALARM_WORD_47 : Word;   // F753 - F768
      ALARM_WORD_48 : Word;   // F769 - F784
      ALARM_WORD_49 : Word;   // F785 - F800
      ALARM_WORD_50 : Word;   // F801 - F816
      ALARM_WORD_51 : Word;   // F817 - F832
      ALARM_WORD_52 : Word;   // F833 - F848
      ALARM_WORD_53 : Word;   // F849 - F864
      ALARM_WORD_54 : Word;   // F865 - F880
      ALARM_WORD_55 : Word;   // F881 - F896
      ALARM_WORD_56 : Word;   // F897 - F912
      ALARM_WORD_57 : Word;   // F913 - F928
      ALARM_WORD_58 : Word;   // F929 - F944
      ALARM_WORD_59 : Word;   // F945 - F960
      ALARM_WORD_60 : Word;   // F961 - F976
      ALARM_WORD_61 : Word;   // F977 - F992
      ALARM_WORD_62 : Word;   // F993 - F1008
      ALARM_WORD_63 : Word;   // F1009- F1024
   END_VAR
BEGIN
END_DATA_BLOCK

DATA_BLOCK "KYD"   // DB200
{ S7_Optimized_Access := 'FALSE' }
VERSION : 0.0
// --------------------------------------------------------------------------------
//     program     :    KYD
//     description :    define all KYD values       
//     name        :    G. Eibelsh鋟ser
//     date        :    26.10.2007
// 
//     revision    :   
//     name        :   
//     date        :    
// 
//                     (c)PVA TePla AG       
//     --------------------------------------------------------------------------------
   VAR
      MOD_AUTO : Bool;   // word 0
      MOD_MANUAL : Bool;
      MOD_SEMI_AUTO : Bool;
      MOD_START : Bool;
      MOD_CONTINUE : Bool;
      MOD_STOP : Bool;
      KEY_PROCESS : Bool;
      SPARE_0_7 : Bool;
      MOD_PUMP_DOWN : Bool;
      MOD_MELTING : Bool;
      MOD_DIP : Bool;
      MOD_NECK : Bool;
      MOD_SHOULDER : Bool;
      MOD_BODY : Bool;
      MOD_ENDCONE : Bool;
      MOD_REMOVAL : Bool;
      MOD_SHUT_DOWN : Bool;   // word 1
      MOD_EMG_OFF : Bool;
      STATE_STD_BY : Bool;
      STATE_SERV : Bool;
      STATE_RUN : Bool;
      STATE_VAC_TEST : Bool;
      PC_ALIVE : Bool;
      STATE_LOADING : Bool;
      SMI_XT_SPD_ON : Bool;
      SMI_XT_SPD_OFF : Bool;
      SMI_XT_ROT_ON : Bool;
      SMI_XT_ROT_OFF : Bool;
      SMI_CR_SPD_ON : Bool;
      SMI_CR_SPD_OFF : Bool;
      SMI_CR_ROT_ON : Bool;
      SMI_CR_ROT_OFF : Bool;
      SMI_HTR_1_ON : Bool;   // word 2
      SMI_HTR_1_OFF : Bool;
      SMI_HTR_2_ON : Bool;
      SMI_HTR_2_OFF : Bool;
      SMI_GAS_FLW_ON : Bool;
      SMI_GAS_FLW_OFF : Bool;
      SMI_GAS_PRS_ON : Bool;
      SMI_GAS_PRS_OFF : Bool;
      SMI_SI_FDR_ON : Bool;
      SMI_SI_FDR_OFF : Bool;
      SMI_DOP_FDR_ON : Bool;
      SMI_DOP_FDR_OFF : Bool;
      SMI_MAG_ON : Bool;
      SMI_MAG_OFF : Bool;
      SMI_CR_SPD_COF_ON : Bool;
      SMI_CR_SPD_COF_OFF : Bool;
      PRS_CTRL_RST : Bool;   // word 3
      DIA_CTRL_RST : Bool;
      HTR_1_CTRL_RST : Bool;
      SPD_CTRL_RST : Bool;
      CRUC_ROT_CTRL_RST : Bool;
      MLT_TMP_CTRL_RST : Bool;
      GRW_RTE_CTRL_RST : Bool;
      MLT_DRIFT_CTRL_RST : Bool;
      XT_LFT_UP : Bool;
      XT_LFT_DN : Bool;
      XT_LFT_OFF : Bool;
      XT_LFT_FST : Bool;
      XT_ROT_CW : Bool;
      XT_ROT_CCW : Bool;
      XT_ROT_OFF : Bool;
      TAR_XT_WGT_CELL : Bool;
      CR_LFT_UP : Bool;   // word 4
      CR_LFT_DN : Bool;
      CR_LFT_OFF : Bool;
      CR_LFT_FST : Bool;
      CR_ROT_CW : Bool;
      CR_ROT_CCW : Bool;
      CR_ROT_OFF : Bool;
      TAR_FDR_WGT_CELL : Bool;
      HTR_1_ON : Bool;
      HTR_1_OFF : Bool;
      CTL_HTR_1_TMP_ON : Bool;
      CTL_HTR_1_TMP_OFF : Bool;
      HTR_2_ON : Bool;
      HTR_2_OFF : Bool;
      CTL_HTR_2_TMP_ON : Bool;
      CTL_HTR_2_TMP_OFF : Bool;
      MAG_ON : Bool;   // word 5
      MAG_OFF : Bool;
      V24_OP : Bool;
      V24_CL : Bool;
      V3_2_OP : Bool;
      V3_2_CL : Bool;
      V15_OPEN : Bool;
      V15_CLOSE : Bool;
      CTL_PRS_ON : Bool;
      CTL_PRS_OFF : Bool;
      V1_OPEN_REQ : Bool;
      V1_CLOSE_REQ : Bool;
      V2_1_OPEN : Bool;
      V2_1_CLOSE : Bool;
      V3_OPEN : Bool;
      V3_CLOSE : Bool;
      V4_OPEN : Bool;   // word 6
      V4_CLOSE : Bool;
      V5_OPEN : Bool;
      V5_CLOSE : Bool;
      V6_OPEN : Bool;
      V6_CLOSE : Bool;
      V8_OPEN : Bool;
      V8_CLOSE : Bool;
      V11_OPEN : Bool;
      V11_CLOSE : Bool;
      V12_OPEN : Bool;
      V12_CLOSE : Bool;
      V2_2_OPEN : Bool;
      V2_2_CLOSE : Bool;
      V9_1_OPEN : Bool;
      V9_1_CLOSE : Bool;
      V9_2_OPEN : Bool;   // word 7
      V9_2_CLOSE : Bool;
      V16_1_OPEN : Bool;
      V16_1_CLOSE : Bool;
      V16_2_OPEN : Bool;
      V16_2_CLOSE : Bool;
      V21_OPEN : Bool;
      V21_CLOSE : Bool;
      P1_ON : Bool;
      P1_OFF : Bool;
      P3_ON : Bool;
      P3_OFF : Bool;
      SPARE_15_4 : Bool;
      V2_1_SEL : Bool;
      V2_2_SEL : Bool;
      V2_X_SEL : Bool;
      MCC_ON : Bool;   // word 8
      MCC_OFF : Bool;
      MCC_TST_ON : Bool;
      MCC_TST_OFF : Bool;
      LSR_ON : Bool;
      LSR_OFF : Bool;
      LSR_FIL_LOW : Bool;
      LSR_FIL_HI : Bool;
      CAM_OFF : Bool;
      CAM_MLT : Bool;
      CAM_DIP : Bool;
      CAM_DIA : Bool;
      CAM_CAL : Bool;
      CAM_SEL_1 : Bool;
      CAM_SEL_2 : Bool;
      CAM_RST_THR_ADJ : Bool;
      ALARM_ACKN : Bool;   // word 9
      DIP2 : Bool;
      DIP2_NEW_LEN : Bool;
      ENDCONE_NO_SD : Bool;
      MOVE_CR_FOR_DIP : Bool;
      ALM_SND : Bool;
      OP_CALL_ON : Bool;
      OP_CALL_OFF : Bool;
      OP_CALL_ACK : Bool;
      OP_XT_DRP_OUT_PRT : Bool;
      CL_XT_DRP_OUT_PRT : Bool;
      FDR_TUBE_DRV_IN : Bool;
      FDR_TUBE_DRV_OUT : Bool;
      FDR_TUBE_DRV_OFF : Bool;
      FDR_FLP_CTL_ON : Bool;
      FDR_FLP_CTL_OFF : Bool;
      XT_LFT_TRIP_RES : Bool;   // word 10
      XT_ROT_TRIP_RES : Bool;
      CR_LFT_TRIP_RES : Bool;
      CR_ROT_TRIP_RES : Bool;
      CGT_LFT_TRIP_RES : Bool;
      CGT_SWV_TRIP_RES : Bool;
      P2_ON : Bool;
      P2_OFF : Bool;
      CAM_INIT : Bool;
      CAM_ISP_ON : Bool;
      CAM_ISP_OFF : Bool;
      V13_OPEN : Bool;
      V13_CLOSE : Bool;
      V14_OPEN : Bool;
      V14_CLOSE : Bool;
      V17_OPEN : Bool;
      V17_CLOSE : Bool;   // word 11
      V18_OPEN : Bool;
      V18_CLOSE : Bool;
      V19_OPEN : Bool;
      V19_CLOSE : Bool;
      V20_OPEN : Bool;
      V20_CLOSE : Bool;
      V22_OPEN : Bool;
      V22_CLOSE : Bool;
      V23_OPEN : Bool;
      V23_CLOSE : Bool;
      AUX_FIL_ENB : Bool;
      AUX_FIL_DBL : Bool;
      SEL_CAM_PRD_1 : Bool;
      SEL_CAM_PRD_2 : Bool;
      V25_OPEN : Bool;
      V25_CLOSE : Bool;   // word 12
      SI_FIL_FSH_SEQ_ON : Bool;
      SI_FIL_FSH_SEQ_OFF : Bool;
      PD_NEW_LKT : Bool;
      NEW_CARRIER_ID : Bool;
      INGOT_ID_EDIT : Bool;
      LOADING_DONE : Bool;
      MSR_MLT_VIB_ON : Bool;
      RST_SIHI_PU : Bool;
      RST_MLT_LVL : Bool;
      RST_HTR_1_PWR_SPL : Bool;
      RST_HTR_2_PWR_SPL : Bool;
      ACKN_AUTO_OP_CALL : Bool;
      NEXT_MLT_STEP : Bool;
      V25_OP : Bool;
      V25_CL : Bool;
      STATE_MAINTENANCE : Bool;   // word 13
      STATE_ENGINEERING : Bool;
      STATE_BAKE_OUT : Bool;
      SPARE_26_3 : Bool;
      SPARE_26_4 : Bool;
      LSR_SEN_PWR_ON : Bool;
      XT_LFT_REF_RUN : Bool;
      CR_LFT_REF_RUN : Bool;
      TEST_CTRL_ON : Bool;
      TEST_CTRL_OFF : Bool;
      TEST_CTRL_RST : Bool;
      MAG_TRIP_RES : Bool;
      CTL_MLT_DRIFT_ON : Bool;
      CTL_MLT_DRIFT_OFF : Bool;
      MAG_STBY_ON : Bool;
      MAG_STBY_OFF : Bool;
      V3_0_OPEN : Bool;   // word 14
      V3_0_CLOSE : Bool;
      V3_1_OPEN : Bool;
      V3_1_CLOSE : Bool;
      XT_LFT_REF_RESET : Bool;
      CR_LFT_REF_RESET : Bool;
      XT_LFT_REL_LS : Bool;
      CR_LFT_REL_LS : Bool;
      MOB_FDR_DCK_ON : Bool;
      MOB_FDR_UDCK_ON : Bool;
      MOB_FDR_SRV_ON : Bool;
      MOB_FDR_SRV_OFF : Bool;
      MOB_FDR_NEW_LKT : Bool;
      MOB_FDR_IGN_LEAK_RTE : Bool;
      MOB_FDR_ARB_SEQ : Bool;
      MOB_FDR_TUBE_DRV_RES : Bool;
      RE_XT_RMV : Bool;   // word 15
      SPARE_30_1 : Bool;
      SPARE_30_2 : Bool;
      ACC_SC_WTR_STR : Bool;
      ACC_OVP_TEST : Bool;
      MOB_FDR_TUBE_UP : Bool;
      MOB_FDR_TUBE_DN : Bool;
      MOB_FDR_TUBE_STOP : Bool;
      MOB_FDR_MVE_IN_SEQ_ON : Bool;
      MOB_FDR_MVE_OUT_SEQ_ON : Bool;
      MOB_FDR_MVE_SEQ_ARB : Bool;
      MOB_FDR_VIB_ON : Bool;
      MOB_FDR_VIB_OFF : Bool;
      MOB_FDR_CH_SW_R : Bool;
      MOB_FDR_CH_SW_L : Bool;
      MOB_FDR_CH_SW_STOP : Bool;
      CTL_FDG_RTE_ON : Bool;   // word 16
      CTL_FDG_RTE_OFF : Bool;
      CCZ_OP_ON : Bool;
      CCZ_OP_OFF : Bool;
      GAP_CTRL_RST : Bool;
      OFFS_CTRL_RST : Bool;
      EXT_ACQ_TRG : Bool;
      SPARE_32_7 : Bool;
      V7_OP : Bool;
      V7_CL : Bool;
      V7_CLN : Bool;
      VSL_LFT_ENB : Bool;
      VSL_UP : Bool;
      VSL_DN : Bool;
      MAG_DRV_UP : Bool;
      MAG_DRV_DN : Bool;
      SET_HDL_LFT_REF_POS : Bool;   // word 17
      SET_MAG_LFT_REF_POS : Bool;
      BUT_GCH_SWV_IN : Bool;
      BUT_GCH_SWV_OUT : Bool;
      CTL_GAP_ON : Bool;
      CTL_GAP_OFF : Bool;
      SMI_GAP_ON : Bool;
      SMI_GAP_OFF : Bool;
      BEL_LFT_TRIP_RES : Bool;
      TCH_LFT_TRIP_RES : Bool;
      TEC_FLG_LFT_TRIP_RES : Bool;
      FCH_LFT_TRIP_RES : Bool;
      TCH_TILT_TRIP_RES : Bool;
      XT_HDL_LFT_TRIP_RES : Bool;
      XT_HDL_SW_TRIP_RES : Bool;
      V7_LFT_TRIP_RES : Bool;
      V7_SW_TRIP_RES : Bool;
      XT_CLP_ABV_RST : Bool;
      XT_CLP_BLW_RST : Bool;
      EMG : Bool;
      EMG_ENB : Bool;
      XT_EMG_RAI : Bool;
      CR_EMG_LOW : Bool;
      SPARE_36_7 : Bool;
      V3_3_OP : Bool;
      V3_3_CL : Bool;
      V3_4_OP : Bool;
      V3_4_CL : Bool;
      V22_1_OP : Bool;
      V22_1_CL : Bool;
      SPARE_37_6 : Bool;
      SPARE_37_7 : Bool;
      SPARE : Array[38..63] of Byte;
      XT_HDL_SEQ_XT_OUT : Bool;
      XT_HDL_SEQ_LD_CRU : Bool;
      XT_HDL_SEQ_HDL_HZ : Bool;
      XT_HDL_OP_CONT : Bool;
      VSL_HDL_OP_CONT : Bool;
      ABORT_FIL_CLN : Bool;
      MLT_GAP_SEARCH : Bool;
      RESET_ERR_HTR_ETH : Bool;
      V7_LFT_UP : Bool;
      V7_LFT_DN : Bool;
      V7_SW_OUT : Bool;
      V7_SW_IN : Bool;
      SPARE_65_4 : Bool;
      SPARE_65_5 : Bool;
      SPARE_65_6 : Bool;
      SPARE_65_7 : Bool;
      BEL_LFT_UP : Bool;
      BEL_LFT_DN : Bool;
      GCH_LFT_UP : Bool;
      GCH_LFT_DN : Bool;
      GCH_SW_LOCK : Bool;
      GCH_SW_UNLOCK : Bool;
      TCH_LFT_UP : Bool;
      TCH_LFT_DN : Bool;
      TCH_SW_LOCK : Bool;
      TCH_SW_UNLOCK : Bool;
      TCH_TILT_0 : Bool;
      TCH_TILT_30 : Bool;
      TEC_FLG_LFT_UP : Bool;
      TEC_FLG_LFT_DN : Bool;
      TEC_FLG_SW_UNLOCK : Bool;
      UP_FCH_SW_UNLOCK : Bool;
      LO_FCH_SW_UNLOCK : Bool;
      FCH_LFT_UP : Bool;
      FCH_LFT_DN : Bool;
      SPARE68_3 : Bool;
      SPARE68_4 : Bool;
      FCH_HOOK_HOME : Bool;
      FCH_HOOK_WORK : Bool;
      SPARE68_7 : Bool;
      MAG_LFT_UP : Bool;
      MAG_LFT_DN : Bool;
      SPARE_69_2 : Bool;
      TEC_FLG_LFT_REF_SET : Bool;
      FCH_LFT_REF_SET : Bool;
      TEC_FLG_SW_REF_SET : Bool;
      UP_FCH_SW_REF_SET : Bool;
      LO_FCH_SW_REF_SET : Bool;
      XT_HDL_LFT_DN : Bool;
      XT_HDL_LFT_FAST : Bool;
      XT_HDL_LFT_UP : Bool;
      SPARE_70_3 : Bool;
      XT_HDL_SW_OUT : Bool;
      XT_HDL_SW_IN : Bool;
      XT_HDL_SLID_FW : Bool;
      XT_HDL_SLID_BW : Bool;
      XT_DRP_OUT_PRT_OP : Bool;
      XT_DRP_OUT_PRT_CL : Bool;
      XT_CLP_TILT_90 : Bool;
      XT_CLP_TILT_75 : Bool;
      XT_CLP_ABV_OP : Bool;
      XT_CLP_ABV_CL : Bool;
      XT_CLP_BLW_OP : Bool;
      XT_CLP_BLW_CL : Bool;
      XT_HDL_LFT_REF_RES : Bool;
      XT_HDL_LFT_REF_START : Bool;
      XT_NECK_CUT : Bool;
      XT_HDL_LFT_RES : Bool;
      XT_HDL_SW_RES : Bool;
      XT_HDL_SW_REF_START : Bool;
      XT_HDL_SW_REF_RES : Bool;
      XT_HDL_SW_UNLOCK : Bool;
      SPARE_73_0 : Bool;
      SPARE_73_1 : Bool;
      XT_HDL_SW_LOCK : Bool;
      XT_HDL_CLP_OP_CONT : Bool;
      XT_HDL_CUT_OP_CONT : Bool;
      XT_CLP_WGT_TAR : Bool;
      SPARE_73_6 : Bool;
      SPARE_73_7 : Bool;
      HOI_TOOL_CRU_INS : Bool;
      LD_CRU_OP_CONT : Bool;
      LD_CRU_FIN : Bool;
      HOI_TOOL_UNIS : Bool;
      HOI_TOOL_HZ_INS : Bool;
      LD_HZ_OP_CONT : Bool;
      LD_HZ_FIN : Bool;
      SI_FIL_DPD : Bool;
      SPARE_75_0 : Bool;
      SPARE_75_1 : Bool;
      SPARE_75_2 : Bool;
      SPARE_75_3 : Bool;
      SPARE_75_4 : Bool;
      SPARE_75_5 : Bool;
      SPARE_75_6 : Bool;
      SPARE_75_7 : Bool;
      SPARE_OP : Array[76..127] of Byte;
   END_VAR
BEGIN
END_DATA_BLOCK

